LIN {X 0,Y 354.82,Z 396.284,A -85,B 0,C 180,E1 -13539.425,E2 -13539.425} C_VEL
LIN {X 0,Y 354.8,Z 396.287,A -85,B 0,C 180,E1 -13542.871,E2 -13542.871} C_VEL
LIN {X 0,Y 354.764,Z 396.297,A -85,B 0,C 180,E1 -13546.105,E2 -13546.105} C_VEL
LIN {X 0,Y 354.786,Z 396.288,A -85,B 0,C 180,E1 -13549.18,E2 -13549.18} C_VEL
LIN {X 0,Y 354.807,Z 396.289,A -85,B 0,C 180,E1 -13552.403,E2 -13552.403} C_VEL
LIN {X 0,Y 354.811,Z 396.285,A -85,B 0,C 180,E1 -13554.942,E2 -13554.942} C_VEL
LIN {X 0,Y 354.793,Z 396.29,A -85,B 0,C 180,E1 -13558.406,E2 -13558.406} C_VEL
LIN {X 0,Y 354.847,Z 396.283,A -85,B 0,C 180,E1 -13561.62,E2 -13561.62} C_VEL
LIN {X 0,Y 354.9,Z 396.278,A -85,B 0,C 180,E1 -13564.174,E2 -13564.174} C_VEL
LIN {X 0,Y 354.836,Z 396.288,A -85,B 0,C 180,E1 -13567.895,E2 -13567.895} C_VEL
LIN {X 0,Y 354.925,Z 396.277,A -85,B 0,C 180,E1 -13571.892,E2 -13571.892} C_VEL
LIN {X 0,Y 354.945,Z 396.274,A -85,B 0,C 180,E1 -13575.982,E2 -13575.982} C_VEL
LIN {X 0,Y 354.981,Z 396.27,A -85,B 0,C 180,E1 -13579.736,E2 -13579.736} C_VEL
LIN {X 0,Y 355.117,Z 396.251,A -85,B 0,C 180,E1 -13582.037,E2 -13582.037} C_VEL
LIN {X 0,Y 355.095,Z 396.251,A -85,B 0,C 180,E1 -13584.321,E2 -13584.321} C_VEL
LIN {X 0,Y 355.123,Z 396.247,A -85,B 0,C 180,E1 -13588.866,E2 -13588.866} C_VEL
LIN {X 0,Y 354.261,Z 396.361,A -85,B 0,C 180,E1 -13591.137,E2 -13591.137} C_VEL
LIN {X 0,Y 354.367,Z 399.159,A -85,B 0,C 180,E1 -13594.55,E2 -13594.55} C_VEL
LIN {X 0,Y 354.171,Z 402.38,A -85,B 0,C 180,E1 -13597.985,E2 -13597.985} C_VEL
LIN {X 0,Y 353.989,Z 406.197,A -85,B 0,C 180,E1 -13601.887,E2 -13601.887} C_VEL
LIN {X 0,Y 357.569,Z 419.481,A -85,B 0,C 180,E1 -13602.63,E2 -13602.63} C_VEL
LIN {X 0,Y 360.42,Z 432.028,A -85,B 0,C 180,E1 -13603.532,E2 -13603.532} C_VEL
LIN {X 0,Y 360.675,Z 435.61,A -85,B 0,C 180,E1 -13603.81,E2 -13603.81} C_VEL
LIN {X 0,Y 359.83,Z 446.641,A -85,B 0,C 180,E1 -13604.709,E2 -13604.709} C_VEL
LIN {X 0,Y 358.918,Z 456.939,A -85,B 0,C 180,E1 -13605.765,E2 -13605.765} C_VEL
LIN {X 0,Y 357.825,Z 467.606,A -85,B 0,C 180,E1 -13607.134,E2 -13607.134} C_VEL
LIN {X 0,Y 356.806,Z 477.084,A -85,B 0,C 180,E1 -13608.646,E2 -13608.646} C_VEL
LIN {X 0,Y 355.86,Z 485.097,A -85,B 0,C 180,E1 -13610.219,E2 -13610.219} C_VEL
LIN {X 0,Y 355.001,Z 492.665,A -85,B 0,C 180,E1 -13612.095,E2 -13612.095} C_VEL
LIN {X 0,Y 354.467,Z 497.998,A -85,B 0,C 180,E1 -13613.763,E2 -13613.763} C_VEL
LIN {X 0,Y 353.942,Z 503.231,A -85,B 0,C 180,E1 -13615.902,E2 -13615.902} C_VEL
LIN {X 0,Y 353.764,Z 505.535,A -85,B 0,C 180,E1 -13617.189,E2 -13617.189} C_VEL
LIN {X 0,Y 353.425,Z 507.859,A -85,B 0,C 180,E1 -13618.959,E2 -13618.959} C_VEL
LIN {X 0,Y 353.286,Z 509.399,A -85,B 0,C 180,E1 -13621.194,E2 -13621.194} C_VEL
LIN {X 0,Y 353.305,Z 509.409,A -85,B 0,C 180,E1 -13623.334,E2 -13623.334} C_VEL
LIN {X 0,Y 353.494,Z 508.102,A -85,B 0,C 180,E1 -13625.398,E2 -13625.398} C_VEL
LIN {X 0,Y 353.871,Z 505.571,A -85,B 0,C 180,E1 -13627.399,E2 -13627.399} C_VEL
LIN {X 0,Y 354.373,Z 501.731,A -85,B 0,C 180,E1 -13629.392,E2 -13629.392} C_VEL
LIN {X 0,Y 354.911,Z 496.973,A -85,B 0,C 180,E1 -13631.194,E2 -13631.194} C_VEL
LIN {X 0,Y 355.686,Z 490.73,A -85,B 0,C 180,E1 -13633.022,E2 -13633.022} C_VEL
LIN {X 0,Y 356.677,Z 482.905,A -85,B 0,C 180,E1 -13634.832,E2 -13634.832} C_VEL
LIN {X 0,Y 356.532,Z 479.281,A -85,B 0,C 180,E1 -13635.576,E2 -13635.576} C_VEL
LIN {X 0,Y 354.521,Z 473.127,A -85,B 0,C 180,E1 -13636.799,E2 -13636.799} C_VEL
LIN {X 0,Y 352.549,Z 466.534,A -85,B 0,C 180,E1 -13637.955,E2 -13637.955} C_VEL
LIN {X 0,Y 352.45,Z 462.072,A -85,B 0,C 180,E1 -13638.582,E2 -13638.582} C_VEL
LIN {X 0,Y 353.487,Z 452.087,A -85,B 0,C 180,E1 -13639.726,E2 -13639.726} C_VEL
LIN {X 0,Y 354.57,Z 440.766,A -85,B 0,C 180,E1 -13640.757,E2 -13640.757} C_VEL
LIN {X 0,Y 354.763,Z 436.437,A -85,B 0,C 180,E1 -13641.097,E2 -13641.097} C_VEL
LIN {X 0,Y 352.322,Z 425.509,A -85,B 0,C 180,E1 -13642.011,E2 -13642.011} C_VEL
LIN {X 0,Y 348.485,Z 412.951,A -85,B 0,C 180,E1 -13642.905,E2 -13642.905} C_VEL
LIN {X 0,Y 346.967,Z 408.125,A -85,B 0,C 180,E1 -13643.215,E2 -13643.215} C_VEL
LIN {X 0,Y 347.163,Z 405.007,A -85,B 0,C 180,E1 -13646.866,E2 -13646.866} C_VEL
LIN {X 0,Y 347.352,Z 402.017,A -85,B 0,C 180,E1 -13650.46,E2 -13650.46} C_VEL
LIN {X 0,Y 347.472,Z 399.497,A -85,B 0,C 180,E1 -13653.578,E2 -13653.578} C_VEL
LIN {X 0,Y 347.611,Z 397.471,A -85,B 0,C 180,E1 -13656.149,E2 -13656.149} C_VEL
LIN {X 0,Y 347.759,Z 397.173,A -85,B 0,C 180,E1 -13658.668,E2 -13658.668} C_VEL
LIN {X 0,Y 347.862,Z 397.155,A -85,B 0,C 180,E1 -13662.359,E2 -13662.359} C_VEL
LIN {X 0,Y 347.894,Z 397.153,A -85,B 0,C 180,E1 -13665.97,E2 -13665.97} C_VEL
LIN {X 0,Y 347.924,Z 397.149,A -85,B 0,C 180,E1 -13669.525,E2 -13669.525} C_VEL
LIN {X 0,Y 348.087,Z 397.126,A -85,B 0,C 180,E1 -13673.042,E2 -13673.042} C_VEL
LIN {X 0,Y 348.203,Z 397.11,A -85,B 0,C 180,E1 -13677.686,E2 -13677.686} C_VEL
LIN {X 0,Y 348.341,Z 397.092,A -85,B 0,C 180,E1 -13680,E2 -13680} C_VEL
LIN {X 0,Y 348.203,Z 397.109,A -85,B 0,C 180,E1 -13682.313,E2 -13682.313} C_VEL
LIN {X 0,Y 348.087,Z 397.127,A -85,B 0,C 180,E1 -13686.958,E2 -13686.958} C_VEL
LIN {X 0,Y 347.924,Z 397.143,A -85,B 0,C 180,E1 -13690.474,E2 -13690.474} C_VEL
LIN {X 0,Y 347.894,Z 397.15,A -85,B 0,C 180,E1 -13694.15,E2 -13694.15} C_VEL
LIN {X 0,Y 347.887,Z 397.15,A -85,B 0,C 180,E1 -13698.291,E2 -13698.291} C_VEL
LIN {X 0,Y 347.784,Z 397.165,A -85,B 0,C 180,E1 -13701.635,E2 -13701.635} C_VEL
LIN {X 0,Y 347.808,Z 397.162,A -85,B 0,C 180,E1 -13705.109,E2 -13705.109} C_VEL
LIN {X 0,Y 347.804,Z 397.163,A -85,B 0,C 180,E1 -13707.694,E2 -13707.694} C_VEL
LIN {X 0,Y 347.745,Z 397.172,A -85,B 0,C 180,E1 -13710.348,E2 -13710.348} C_VEL
LIN {X 0,Y 347.745,Z 397.174,A -85,B 0,C 180,E1 -13714.044,E2 -13714.044} C_VEL
LIN {X 0,Y 347.76,Z 397.17,A -85,B 0,C 180,E1 -13717.321,E2 -13717.321} C_VEL
LIN {X 0,Y 347.753,Z 397.169,A -85,B 0,C 180,E1 -13720.294,E2 -13720.294} C_VEL
LIN {X 0,Y 347.79,Z 397.314,A -85,B 0,C 180,E1 -13721.824,E2 -13721.824} C_VEL
LIN {X 0,Y 348.52,Z 401.454,A -85,B 0,C 180,E1 -13725.108,E2 -13725.108} C_VEL
LIN {X 0,Y 349.367,Z 406.016,A -85,B 0,C 180,E1 -13728.407,E2 -13728.407} C_VEL
LIN {X 0,Y 350.163,Z 410.733,A -85,B 0,C 180,E1 -13731.524,E2 -13731.524} C_VEL
LIN {X 0,Y 350.496,Z 413.638,A -85,B 0,C 180,E1 -13733.328,E2 -13733.328} C_VEL
LIN {X 0,Y 350.032,Z 417.928,A -85,B 0,C 180,E1 -13735.793,E2 -13735.793} C_VEL
LIN {X 0,Y 349.088,Z 425.333,A -85,B 0,C 180,E1 -13739.781,E2 -13739.781} C_VEL
LIN {X 0,Y 348.231,Z 432.827,A -85,B 0,C 180,E1 -13743.641,E2 -13743.641} C_VEL
LIN {X 0,Y 347.569,Z 440.436,A -85,B 0,C 180,E1 -13747.407,E2 -13747.407} C_VEL
LIN {X 0,Y 347.384,Z 443.37,A -85,B 0,C 180,E1 -13748.844,E2 -13748.844} C_VEL
LIN {X 0,Y 350.074,Z 457.101,A -85,B 0,C 180,E1 -13749.538,E2 -13749.538} C_VEL
LIN {X 0,Y 351.773,Z 470.332,A -85,B 0,C 180,E1 -13750.4,E2 -13750.4} C_VEL
LIN {X 0,Y 352.9,Z 482.718,A -85,B 0,C 180,E1 -13751.419,E2 -13751.419} C_VEL
LIN {X 0,Y 352.517,Z 489.14,A -85,B 0,C 180,E1 -13752,E2 -13752} C_VEL
LIN {X 0,Y 351.116,Z 500.982,A -85,B 0,C 180,E1 -13753.278,E2 -13753.278} C_VEL
LIN {X 0,Y 350.038,Z 510.242,A -85,B 0,C 180,E1 -13754.523,E2 -13754.523} C_VEL
LIN {X 0,Y 349.027,Z 519.346,A -85,B 0,C 180,E1 -13756.017,E2 -13756.017} C_VEL
LIN {X 0,Y 347.998,Z 527.91,A -85,B 0,C 180,E1 -13757.757,E2 -13757.757} C_VEL
LIN {X 0,Y 347.282,Z 534.815,A -85,B 0,C 180,E1 -13759.506,E2 -13759.506} C_VEL
LIN {X 0,Y 346.735,Z 540.361,A -85,B 0,C 180,E1 -13761.256,E2 -13761.256} C_VEL
LIN {X 0,Y 346.419,Z 544.723,A -85,B 0,C 180,E1 -13763.008,E2 -13763.008} C_VEL
LIN {X 0,Y 346.318,Z 547.047,A -85,B 0,C 180,E1 -13764.176,E2 -13764.176} C_VEL
LIN {X 0,Y 346.271,Z 548.911,A -85,B 0,C 180,E1 -13765.343,E2 -13765.343} C_VEL
LIN {X 0,Y 346.223,Z 551.331,A -85,B 0,C 180,E1 -13767.673,E2 -13767.673} C_VEL
LIN {X 0,Y 346.32,Z 551.953,A -85,B 0,C 180,E1 -13768.837,E2 -13768.837} C_VEL
LIN {X 0,Y 346.35,Z 552.148,A -85,B 0,C 180,E1 -13770,E2 -13770} C_VEL
LIN {X 0,Y 346.339,Z 551.916,A -85,B 0,C 180,E1 -13771.162,E2 -13771.162} C_VEL
LIN {X 0,Y 346.206,Z 550.263,A -85,B 0,C 180,E1 -13773.491,E2 -13773.491} C_VEL
LIN {X 0,Y 346.274,Z 548.811,A -85,B 0,C 180,E1 -13774.656,E2 -13774.656} C_VEL
LIN {X 0,Y 346.344,Z 546.358,A -85,B 0,C 180,E1 -13776.116,E2 -13776.116} C_VEL
LIN {X 0,Y 346.591,Z 541.732,A -85,B 0,C 180,E1 -13778.16,E2 -13778.16} C_VEL
LIN {X 0,Y 347.171,Z 535.476,A -85,B 0,C 180,E1 -13780.202,E2 -13780.202} C_VEL
LIN {X 0,Y 347.811,Z 528.66,A -85,B 0,C 180,E1 -13781.953,E2 -13781.953} C_VEL
LIN {X 0,Y 348.832,Z 520.203,A -85,B 0,C 180,E1 -13783.693,E2 -13783.693} C_VEL
LIN {X 0,Y 349.955,Z 510.721,A -85,B 0,C 180,E1 -13785.251,E2 -13785.251} C_VEL
LIN {X 0,Y 350.873,Z 500.782,A -85,B 0,C 180,E1 -13786.584,E2 -13786.584} C_VEL
LIN {X 0,Y 352.108,Z 490.179,A -85,B 0,C 180,E1 -13787.721,E2 -13787.721} C_VEL
LIN {X 0,Y 352.687,Z 483.789,A -85,B 0,C 180,E1 -13788.291,E2 -13788.291} C_VEL
LIN {X 0,Y 351.491,Z 471.586,A -85,B 0,C 180,E1 -13789.281,E2 -13789.281} C_VEL
LIN {X 0,Y 349.823,Z 458.882,A -85,B 0,C 180,E1 -13790.094,E2 -13790.094} C_VEL
LIN {X 0,Y 347.566,Z 446.078,A -85,B 0,C 180,E1 -13790.71,E2 -13790.71} C_VEL
LIN {X 0,Y 347.366,Z 444.386,A -85,B 0,C 180,E1 -13790.813,E2 -13790.813} C_VEL
LIN {X 0,Y 347.975,Z 436.534,A -85,B 0,C 180,E1 -13794.652,E2 -13794.652} C_VEL
LIN {X 0,Y 348.662,Z 429.282,A -85,B 0,C 180,E1 -13798.273,E2 -13798.273} C_VEL
LIN {X 0,Y 349.314,Z 422.946,A -85,B 0,C 180,E1 -13801.54,E2 -13801.54} C_VEL
LIN {X 0,Y 350.133,Z 417.113,A -85,B 0,C 180,E1 -13804.617,E2 -13804.617} C_VEL
LIN {X 0,Y 350.477,Z 412.823,A -85,B 0,C 180,E1 -13806.982,E2 -13806.982} C_VEL
LIN {X 0,Y 349.931,Z 408.97,A -85,B 0,C 180,E1 -13809.243,E2 -13809.243} C_VEL
LIN {X 0,Y 348.909,Z 403.557,A -85,B 0,C 180,E1 -13812.619,E2 -13812.619} C_VEL
LIN {X 0,Y 348.055,Z 398.681,A -85,B 0,C 180,E1 -13815.843,E2 -13815.843} C_VEL
LIN {X 0,Y 347.778,Z 397.166,A -85,B 0,C 180,E1 -13817.036,E2 -13817.036} C_VEL
LIN {X 0,Y 347.761,Z 397.168,A -85,B 0,C 180,E1 -13821.208,E2 -13821.208} C_VEL
LIN {X 0,Y 347.783,Z 397.161,A -85,B 0,C 180,E1 -13824.124,E2 -13824.124} C_VEL
LIN {X 0,Y 347.732,Z 397.167,A -85,B 0,C 180,E1 -13828.086,E2 -13828.086} C_VEL
LIN {X 0,Y 347.772,Z 397.167,A -85,B 0,C 180,E1 -13830.987,E2 -13830.987} C_VEL
LIN {X 0,Y 347.824,Z 397.156,A -85,B 0,C 180,E1 -13833.607,E2 -13833.607} C_VEL
LIN {X 0,Y 347.781,Z 397.161,A -85,B 0,C 180,E1 -13836.161,E2 -13836.161} C_VEL
LIN {X 0,Y 347.805,Z 397.158,A -85,B 0,C 180,E1 -13839.909,E2 -13839.909} C_VEL
LIN {X 0,Y 347.858,Z 397.153,A -85,B 0,C 180,E1 -13842.359,E2 -13842.359} C_VEL
LIN {X 0,Y 347.89,Z 397.147,A -85,B 0,C 180,E1 -13845.971,E2 -13845.971} C_VEL
LIN {X 0,Y 347.921,Z 397.144,A -85,B 0,C 180,E1 -13849.525,E2 -13849.525} C_VEL
LIN {X 0,Y 348.084,Z 397.126,A -85,B 0,C 180,E1 -13853.042,E2 -13853.042} C_VEL
LIN {X 0,Y 348.2,Z 397.109,A -85,B 0,C 180,E1 -13857.687,E2 -13857.687} C_VEL
LIN {X 0,Y 348.36,Z 397.09,A -85,B 0,C 180,E1 -13860,E2 -13860} C_VEL
LIN {X 0,Y 348.2,Z 397.112,A -85,B 0,C 180,E1 -13862.314,E2 -13862.314} C_VEL
LIN {X 0,Y 348.098,Z 397.124,A -85,B 0,C 180,E1 -13866.958,E2 -13866.958} C_VEL
LIN {X 0,Y 347.96,Z 397.139,A -85,B 0,C 180,E1 -13869.299,E2 -13869.299} C_VEL
LIN {X 0,Y 347.882,Z 397.151,A -85,B 0,C 180,E1 -13872.84,E2 -13872.84} C_VEL
LIN {X 0,Y 347.832,Z 397.16,A -85,B 0,C 180,E1 -13876.432,E2 -13876.432} C_VEL
LIN {X 0,Y 347.849,Z 397.154,A -85,B 0,C 180,E1 -13878.861,E2 -13878.861} C_VEL
LIN {X 0,Y 347.767,Z 397.167,A -85,B 0,C 180,E1 -13882.58,E2 -13882.58} C_VEL
LIN {X 0,Y 347.806,Z 397.158,A -85,B 0,C 180,E1 -13885.109,E2 -13885.109} C_VEL
LIN {X 0,Y 347.805,Z 397.159,A -85,B 0,C 180,E1 -13887.695,E2 -13887.695} C_VEL
LIN {X 0,Y 347.758,Z 397.169,A -85,B 0,C 180,E1 -13890.347,E2 -13890.347} C_VEL
LIN {X 0,Y 347.739,Z 397.17,A -85,B 0,C 180,E1 -13894.465,E2 -13894.465} C_VEL
LIN {X 0,Y 347.772,Z 397.166,A -85,B 0,C 180,E1 -13897.99,E2 -13897.99} C_VEL
LIN {X 0,Y 347.763,Z 397.166,A -85,B 0,C 180,E1 -13901.829,E2 -13901.829} C_VEL
LIN {X 0,Y 347.704,Z 397.17,A -85,B 0,C 180,E1 -13905.027,E2 -13905.027} C_VEL
LIN {X 0,Y 347.748,Z 397.168,A -85,B 0,C 180,E1 -13908.398,E2 -13908.398} C_VEL
LIN {X 0,Y 347.773,Z 397.167,A -85,B 0,C 180,E1 -13912.012,E2 -13912.012} C_VEL
LIN {X 0,Y 347.743,Z 397.167,A -85,B 0,C 180,E1 -13915.537,E2 -13915.537} C_VEL
LIN {X 0,Y 347.745,Z 397.169,A -85,B 0,C 180,E1 -13918.301,E2 -13918.301} C_VEL
LIN {X 0,Y 347.778,Z 397.161,A -85,B 0,C 180,E1 -13920.989,E2 -13920.989} C_VEL
LIN {X 0,Y 347.832,Z 397.157,A -85,B 0,C 180,E1 -13923.609,E2 -13923.609} C_VEL
LIN {X 0,Y 347.79,Z 397.164,A -85,B 0,C 180,E1 -13926.163,E2 -13926.163} C_VEL
LIN {X 0,Y 347.819,Z 397.162,A -85,B 0,C 180,E1 -13929.91,E2 -13929.91} C_VEL
LIN {X 0,Y 347.869,Z 397.152,A -85,B 0,C 180,E1 -13932.36,E2 -13932.36} C_VEL
LIN {X 0,Y 347.9,Z 397.151,A -85,B 0,C 180,E1 -13935.971,E2 -13935.971} C_VEL
LIN {X 0,Y 347.931,Z 397.145,A -85,B 0,C 180,E1 -13939.526,E2 -13939.526} C_VEL
LIN {X 0,Y 348.078,Z 397.129,A -85,B 0,C 180,E1 -13941.875,E2 -13941.875} C_VEL
LIN {X 0,Y 348.07,Z 397.127,A -85,B 0,C 180,E1 -13944.206,E2 -13944.206} C_VEL
LIN {X 0,Y 348.091,Z 397.122,A -85,B 0,C 180,E1 -13948.843,E2 -13948.843} C_VEL
LIN {X 0,Y 347.206,Z 397.239,A -85,B 0,C 180,E1 -13951.16,E2 -13951.16} C_VEL
LIN {X 0,Y 347.316,Z 400.101,A -85,B 0,C 180,E1 -13954.643,E2 -13954.643} C_VEL
LIN {X 0,Y 347.111,Z 403.298,A -85,B 0,C 180,E1 -13958.148,E2 -13958.148} C_VEL
LIN {X 0,Y 346.894,Z 406.47,A -85,B 0,C 180,E1 -13961.467,E2 -13961.467} C_VEL
LIN {X 0,Y 350.716,Z 420.405,A -85,B 0,C 180,E1 -13962.293,E2 -13962.293} C_VEL
LIN {X 0,Y 353.52,Z 432.875,A -85,B 0,C 180,E1 -13963.216,E2 -13963.216} C_VEL
LIN {X 0,Y 353.9,Z 436.266,A -85,B 0,C 180,E1 -13963.494,E2 -13963.494} C_VEL
LIN {X 0,Y 353.014,Z 447.259,A -85,B 0,C 180,E1 -13964.41,E2 -13964.41} C_VEL
LIN {X 0,Y 351.922,Z 458.801,A -85,B 0,C 180,E1 -13965.64,E2 -13965.64} C_VEL
LIN {X 0,Y 350.819,Z 468.918,A -85,B 0,C 180,E1 -13966.992,E2 -13966.992} C_VEL
LIN {X 0,Y 349.859,Z 477.746,A -85,B 0,C 180,E1 -13968.444,E2 -13968.444} C_VEL
LIN {X 0,Y 348.897,Z 485.606,A -85,B 0,C 180,E1 -13970.025,E2 -13970.025} C_VEL
LIN {X 0,Y 348.058,Z 492.489,A -85,B 0,C 180,E1 -13971.745,E2 -13971.745} C_VEL
LIN {X 0,Y 347.531,Z 497.324,A -85,B 0,C 180,E1 -13973.225,E2 -13973.225} C_VEL
LIN {X 0,Y 346.998,Z 502.312,A -85,B 0,C 180,E1 -13975.171,E2 -13975.171} C_VEL
LIN {X 0,Y 346.738,Z 505.624,A -85,B 0,C 180,E1 -13976.895,E2 -13976.895} C_VEL
LIN {X 0,Y 346.321,Z 508.605,A -85,B 0,C 180,E1 -13979.236,E2 -13979.236} C_VEL
LIN {X 0,Y 346.208,Z 509.906,A -85,B 0,C 180,E1 -13981.504,E2 -13981.504} C_VEL
LIN {X 0,Y 346.232,Z 509.74,A -85,B 0,C 180,E1 -13983.67,E2 -13983.67} C_VEL
LIN {X 0,Y 346.525,Z 508.021,A -85,B 0,C 180,E1 -13986.026,E2 -13986.026} C_VEL
LIN {X 0,Y 346.898,Z 505.598,A -85,B 0,C 180,E1 -13987.802,E2 -13987.802} C_VEL
LIN {X 0,Y 347.388,Z 501.733,A -85,B 0,C 180,E1 -13989.755,E2 -13989.755} C_VEL
LIN {X 0,Y 348.058,Z 496.267,A -85,B 0,C 180,E1 -13991.784,E2 -13991.784} C_VEL
LIN {X 0,Y 349.014,Z 489.379,A -85,B 0,C 180,E1 -13993.74,E2 -13993.74} C_VEL
LIN {X 0,Y 349.993,Z 482.21,A -85,B 0,C 180,E1 -13995.346,E2 -13995.346} C_VEL
LIN {X 0,Y 351.09,Z 473.823,A -85,B 0,C 180,E1 -13996.876,E2 -13996.876} C_VEL
LIN {X 0,Y 352.297,Z 463.334,A -85,B 0,C 180,E1 -13998.424,E2 -13998.424} C_VEL
LIN {X 0,Y 352.45,Z 462.072,A -85,B 0,C 180,E1 -13998.582,E2 -13998.582} C_VEL
LIN {X 0,Y 352.394,Z 455.899,A -85,B 0,C 180,E1 -13999.362,E2 -13999.362} C_VEL
LIN {X 0,Y 351.186,Z 449.734,A -85,B 0,C 180,E1 -14000.13,E2 -14000.13} C_VEL
LIN {X 0,Y 349.464,Z 443.357,A -85,B 0,C 180,E1 -14000.867,E2 -14000.867} C_VEL
LIN {X 0,Y 347.859,Z 436.701,A -85,B 0,C 180,E1 -14001.543,E2 -14001.543} C_VEL
LIN {X 0,Y 345.286,Z 425.748,A -85,B 0,C 180,E1 -14002.489,E2 -14002.489} C_VEL
LIN {X 0,Y 341.446,Z 413.364,A -85,B 0,C 180,E1 -14003.4,E2 -14003.4} C_VEL
LIN {X 0,Y 339.942,Z 408.589,A -85,B 0,C 180,E1 -14003.734,E2 -14003.734} C_VEL
LIN {X 0,Y 340.147,Z 405.423,A -85,B 0,C 180,E1 -14007.506,E2 -14007.506} C_VEL
LIN {X 0,Y 340.306,Z 403.155,A -85,B 0,C 180,E1 -14010.287,E2 -14010.287} C_VEL
LIN {X 0,Y 340.436,Z 401.017,A -85,B 0,C 180,E1 -14012.988,E2 -14012.988} C_VEL
LIN {X 0,Y 340.612,Z 398.955,A -85,B 0,C 180,E1 -14015.627,E2 -14015.627} C_VEL
LIN {X 0,Y 340.58,Z 398.068,A -85,B 0,C 180,E1 -14016.916,E2 -14016.916} C_VEL
LIN {X 0,Y 340.782,Z 398.039,A -85,B 0,C 180,E1 -14020.733,E2 -14020.733} C_VEL
LIN {X 0,Y 340.782,Z 398.038,A -85,B 0,C 180,E1 -14023.218,E2 -14023.218} C_VEL
LIN {X 0,Y 340.84,Z 398.03,A -85,B 0,C 180,E1 -14026.89,E2 -14026.89} C_VEL
LIN {X 0,Y 340.91,Z 398.02,A -85,B 0,C 180,E1 -14030.507,E2 -14030.507} C_VEL
LIN {X 0,Y 341.055,Z 398.001,A -85,B 0,C 180,E1 -14032.898,E2 -14032.898} C_VEL
LIN {X 0,Y 341.165,Z 397.986,A -85,B 0,C 180,E1 -14037.639,E2 -14037.639} C_VEL
LIN {X 0,Y 341.291,Z 397.97,A -85,B 0,C 180,E1 -14040,E2 -14040} C_VEL
LIN {X 0,Y 341.165,Z 397.986,A -85,B 0,C 180,E1 -14042.361,E2 -14042.361} C_VEL
LIN {X 0,Y 341.055,Z 398.003,A -85,B 0,C 180,E1 -14047.102,E2 -14047.102} C_VEL
LIN {X 0,Y 340.866,Z 398.022,A -85,B 0,C 180,E1 -14050.694,E2 -14050.694} C_VEL
LIN {X 0,Y 340.859,Z 398.026,A -85,B 0,C 180,E1 -14054.325,E2 -14054.325} C_VEL
LIN {X 0,Y 340.834,Z 398.027,A -85,B 0,C 180,E1 -14058.467,E2 -14058.467} C_VEL
LIN {X 0,Y 340.75,Z 398.042,A -85,B 0,C 180,E1 -14061.857,E2 -14061.857} C_VEL
LIN {X 0,Y 340.768,Z 398.039,A -85,B 0,C 180,E1 -14065.665,E2 -14065.665} C_VEL
LIN {X 0,Y 340.725,Z 398.043,A -85,B 0,C 180,E1 -14068.321,E2 -14068.321} C_VEL
LIN {X 0,Y 340.694,Z 398.047,A -85,B 0,C 180,E1 -14071.045,E2 -14071.045} C_VEL
LIN {X 0,Y 340.715,Z 398.047,A -85,B 0,C 180,E1 -14075.279,E2 -14075.279} C_VEL
LIN {X 0,Y 340.715,Z 398.047,A -85,B 0,C 180,E1 -14078.388,E2 -14078.388} C_VEL
LIN {X 0,Y 340.724,Z 398.137,A -85,B 0,C 180,E1 -14081.159,E2 -14081.159} C_VEL
LIN {X 0,Y 341.408,Z 402.065,A -85,B 0,C 180,E1 -14084.419,E2 -14084.419} C_VEL
LIN {X 0,Y 342.238,Z 406.375,A -85,B 0,C 180,E1 -14087.67,E2 -14087.67} C_VEL
LIN {X 0,Y 343.082,Z 411.395,A -85,B 0,C 180,E1 -14091.117,E2 -14091.117} C_VEL
LIN {X 0,Y 343.476,Z 414.258,A -85,B 0,C 180,E1 -14092.939,E2 -14092.939} C_VEL
LIN {X 0,Y 343.222,Z 417.737,A -85,B 0,C 180,E1 -14095.017,E2 -14095.017} C_VEL
LIN {X 0,Y 342.181,Z 425.051,A -85,B 0,C 180,E1 -14099.105,E2 -14099.105} C_VEL
LIN {X 0,Y 341.275,Z 432.497,A -85,B 0,C 180,E1 -14103.06,E2 -14103.06} C_VEL
LIN {X 0,Y 340.547,Z 440.057,A -85,B 0,C 180,E1 -14106.914,E2 -14106.914} C_VEL
LIN {X 0,Y 340.373,Z 443.137,A -85,B 0,C 180,E1 -14108.351,E2 -14108.351} C_VEL
LIN {X 0,Y 343.09,Z 456.301,A -85,B 0,C 180,E1 -14109.044,E2 -14109.044} C_VEL
LIN {X 0,Y 344.841,Z 469.313,A -85,B 0,C 180,E1 -14109.915,E2 -14109.915} C_VEL
LIN {X 0,Y 345.836,Z 481.465,A -85,B 0,C 180,E1 -14110.927,E2 -14110.927} C_VEL
LIN {X 0,Y 346.083,Z 485.84,A -85,B 0,C 180,E1 -14111.347,E2 -14111.347} C_VEL
LIN {X 0,Y 344.767,Z 497.117,A -85,B 0,C 180,E1 -14112.502,E2 -14112.502} C_VEL
LIN {X 0,Y 343.435,Z 507.636,A -85,B 0,C 180,E1 -14113.856,E2 -14113.856} C_VEL
LIN {X 0,Y 342.32,Z 517.398,A -85,B 0,C 180,E1 -14115.434,E2 -14115.434} C_VEL
LIN {X 0,Y 341.198,Z 526.29,A -85,B 0,C 180,E1 -14117.207,E2 -14117.207} C_VEL
LIN {X 0,Y 340.342,Z 533.432,A -85,B 0,C 180,E1 -14118.988,E2 -14118.988} C_VEL
LIN {X 0,Y 339.697,Z 539.99,A -85,B 0,C 180,E1 -14121.073,E2 -14121.073} C_VEL
LIN {X 0,Y 339.347,Z 544.336,A -85,B 0,C 180,E1 -14122.862,E2 -14122.862} C_VEL
LIN {X 0,Y 339.238,Z 546.652,A -85,B 0,C 180,E1 -14124.054,E2 -14124.054} C_VEL
LIN {X 0,Y 339.189,Z 548.503,A -85,B 0,C 180,E1 -14125.246,E2 -14125.246} C_VEL
LIN {X 0,Y 339.13,Z 549.906,A -85,B 0,C 180,E1 -14126.435,E2 -14126.435} C_VEL
LIN {X 0,Y 339.227,Z 551.529,A -85,B 0,C 180,E1 -14128.813,E2 -14128.813} C_VEL
LIN {X 0,Y 339.29,Z 551.716,A -85,B 0,C 180,E1 -14130,E2 -14130} C_VEL
LIN {X 0,Y 339.26,Z 551.478,A -85,B 0,C 180,E1 -14131.187,E2 -14131.187} C_VEL
LIN {X 0,Y 339.13,Z 549.815,A -85,B 0,C 180,E1 -14133.564,E2 -14133.564} C_VEL
LIN {X 0,Y 339.193,Z 548.35,A -85,B 0,C 180,E1 -14134.754,E2 -14134.754} C_VEL
LIN {X 0,Y 339.298,Z 545.331,A -85,B 0,C 180,E1 -14136.541,E2 -14136.541} C_VEL
LIN {X 0,Y 339.547,Z 541.243,A -85,B 0,C 180,E1 -14138.33,E2 -14138.33} C_VEL
LIN {X 0,Y 340.14,Z 534.965,A -85,B 0,C 180,E1 -14140.415,E2 -14140.415} C_VEL
LIN {X 0,Y 340.841,Z 528.126,A -85,B 0,C 180,E1 -14142.201,E2 -14142.201} C_VEL
LIN {X 0,Y 341.877,Z 519.627,A -85,B 0,C 180,E1 -14143.977,E2 -14143.977} C_VEL
LIN {X 0,Y 342.966,Z 510.886,A -85,B 0,C 180,E1 -14145.449,E2 -14145.449} C_VEL
LIN {X 0,Y 344.051,Z 500.125,A -85,B 0,C 180,E1 -14146.922,E2 -14146.922} C_VEL
LIN {X 0,Y 345.309,Z 489.46,A -85,B 0,C 180,E1 -14148.081,E2 -14148.081} C_VEL
LIN {X 0,Y 345.774,Z 484.738,A -85,B 0,C 180,E1 -14148.516,E2 -14148.516} C_VEL
LIN {X 0,Y 344.735,Z 473.294,A -85,B 0,C 180,E1 -14149.498,E2 -14149.498} C_VEL
LIN {X 0,Y 342.999,Z 459.609,A -85,B 0,C 180,E1 -14150.42,E2 -14150.42} C_VEL
LIN {X 0,Y 340.7,Z 446.287,A -85,B 0,C 180,E1 -14151.098,E2 -14151.098} C_VEL
LIN {X 0,Y 340.338,Z 444.086,A -85,B 0,C 180,E1 -14151.184,E2 -14151.184} C_VEL
LIN {X 0,Y 340.936,Z 436.673,A -85,B 0,C 180,E1 -14154.905,E2 -14154.905} C_VEL
LIN {X 0,Y 341.732,Z 428.894,A -85,B 0,C 180,E1 -14158.9,E2 -14158.9} C_VEL
LIN {X 0,Y 342.608,Z 421.612,A -85,B 0,C 180,E1 -14162.749,E2 -14162.749} C_VEL
LIN {X 0,Y 343.357,Z 416.262,A -85,B 0,C 180,E1 -14165.685,E2 -14165.685} C_VEL
LIN {X 0,Y 343.317,Z 412.438,A -85,B 0,C 180,E1 -14167.887,E2 -14167.887} C_VEL
LIN {X 0,Y 342.41,Z 407.302,A -85,B 0,C 180,E1 -14171.055,E2 -14171.055} C_VEL
LIN {X 0,Y 341.474,Z 402.196,A -85,B 0,C 180,E1 -14174.407,E2 -14174.407} C_VEL
LIN {X 0,Y 340.731,Z 398.044,A -85,B 0,C 180,E1 -14177.342,E2 -14177.342} C_VEL
LIN {X 0,Y 340.705,Z 398.046,A -85,B 0,C 180,E1 -14180.248,E2 -14180.248} C_VEL
LIN {X 0,Y 340.705,Z 398.043,A -85,B 0,C 180,E1 -14183.558,E2 -14183.558} C_VEL
LIN {X 0,Y 340.686,Z 398.045,A -85,B 0,C 180,E1 -14186.153,E2 -14186.153} C_VEL
LIN {X 0,Y 340.735,Z 398.039,A -85,B 0,C 180,E1 -14190.329,E2 -14190.329} C_VEL
LIN {X 0,Y 340.796,Z 398.035,A -85,B 0,C 180,E1 -14193.019,E2 -14193.019} C_VEL
LIN {X 0,Y 340.749,Z 398.037,A -85,B 0,C 180,E1 -14195.638,E2 -14195.638} C_VEL
LIN {X 0,Y 340.745,Z 398.038,A -85,B 0,C 180,E1 -14199.474,E2 -14199.474} C_VEL
LIN {X 0,Y 340.85,Z 398.024,A -85,B 0,C 180,E1 -14201.984,E2 -14201.984} C_VEL
LIN {X 0,Y 340.862,Z 398.022,A -85,B 0,C 180,E1 -14205.705,E2 -14205.705} C_VEL
LIN {X 0,Y 340.863,Z 398.023,A -85,B 0,C 180,E1 -14209.306,E2 -14209.306} C_VEL
LIN {X 0,Y 341.051,Z 398.003,A -85,B 0,C 180,E1 -14212.898,E2 -14212.898} C_VEL
LIN {X 0,Y 341.162,Z 397.985,A -85,B 0,C 180,E1 -14217.639,E2 -14217.639} C_VEL
LIN {X 0,Y 341.309,Z 397.968,A -85,B 0,C 180,E1 -14220,E2 -14220} C_VEL
LIN {X 0,Y 341.162,Z 397.989,A -85,B 0,C 180,E1 -14222.361,E2 -14222.361} C_VEL
LIN {X 0,Y 341.067,Z 397.998,A -85,B 0,C 180,E1 -14227.102,E2 -14227.102} C_VEL
LIN {X 0,Y 340.863,Z 398.026,A -85,B 0,C 180,E1 -14230.694,E2 -14230.694} C_VEL
LIN {X 0,Y 340.856,Z 398.028,A -85,B 0,C 180,E1 -14234.325,E2 -14234.325} C_VEL
LIN {X 0,Y 340.831,Z 398.032,A -85,B 0,C 180,E1 -14238.467,E2 -14238.467} C_VEL
LIN {X 0,Y 340.747,Z 398.038,A -85,B 0,C 180,E1 -14241.858,E2 -14241.858} C_VEL
LIN {X 0,Y 340.766,Z 398.035,A -85,B 0,C 180,E1 -14245.665,E2 -14245.665} C_VEL
LIN {X 0,Y 340.735,Z 398.044,A -85,B 0,C 180,E1 -14248.32,E2 -14248.32} C_VEL
LIN {X 0,Y 340.698,Z 398.043,A -85,B 0,C 180,E1 -14251.045,E2 -14251.045} C_VEL
LIN {X 0,Y 340.714,Z 398.041,A -85,B 0,C 180,E1 -14255.28,E2 -14255.28} C_VEL
LIN {X 0,Y 340.714,Z 398.045,A -85,B 0,C 180,E1 -14258.389,E2 -14258.389} C_VEL
LIN {X 0,Y 340.726,Z 398.044,A -85,B 0,C 180,E1 -14262.052,E2 -14262.052} C_VEL
LIN {X 0,Y 340.649,Z 398.054,A -85,B 0,C 180,E1 -14266.228,E2 -14266.228} C_VEL
LIN {X 0,Y 340.686,Z 398.047,A -85,B 0,C 180,E1 -14269.754,E2 -14269.754} C_VEL
LIN {X 0,Y 340.704,Z 398.042,A -85,B 0,C 180,E1 -14273.26,E2 -14273.26} C_VEL
LIN {X 0,Y 340.693,Z 398.049,A -85,B 0,C 180,E1 -14276.155,E2 -14276.155} C_VEL
LIN {X 0,Y 340.741,Z 398.04,A -85,B 0,C 180,E1 -14280.33,E2 -14280.33} C_VEL
LIN {X 0,Y 340.804,Z 398.03,A -85,B 0,C 180,E1 -14283.021,E2 -14283.021} C_VEL
LIN {X 0,Y 340.757,Z 398.038,A -85,B 0,C 180,E1 -14285.639,E2 -14285.639} C_VEL
LIN {X 0,Y 340.75,Z 398.038,A -85,B 0,C 180,E1 -14289.475,E2 -14289.475} C_VEL
LIN {X 0,Y 340.86,Z 398.028,A -85,B 0,C 180,E1 -14291.985,E2 -14291.985} C_VEL
LIN {X 0,Y 340.872,Z 398.026,A -85,B 0,C 180,E1 -14295.706,E2 -14295.706} C_VEL
LIN {X 0,Y 340.874,Z 398.022,A -85,B 0,C 180,E1 -14299.307,E2 -14299.307} C_VEL
LIN {X 0,Y 341.079,Z 397.995,A -85,B 0,C 180,E1 -14302.899,E2 -14302.899} C_VEL
LIN {X 0,Y 340.805,Z 398.031,A -85,B 0,C 180,E1 -14305.269,E2 -14305.269} C_VEL
LIN {X 0,Y 341.06,Z 397.998,A -85,B 0,C 180,E1 -14308.82,E2 -14308.82} C_VEL
LIN {X 0,Y 340.151,Z 398.118,A -85,B 0,C 180,E1 -14311.184,E2 -14311.184} C_VEL
LIN {X 0,Y 340.265,Z 401.076,A -85,B 0,C 180,E1 -14314.739,E2 -14314.739} C_VEL
LIN {X 0,Y 340.045,Z 404.282,A -85,B 0,C 180,E1 -14318.319,E2 -14318.319} C_VEL
LIN {X 0,Y 339.852,Z 406.819,A -85,B 0,C 180,E1 -14321.066,E2 -14321.066} C_VEL
LIN {X 0,Y 343.707,Z 420.886,A -85,B 0,C 180,E1 -14321.911,E2 -14321.911} C_VEL
LIN {X 0,Y 346.261,Z 431.812,A -85,B 0,C 180,E1 -14322.737,E2 -14322.737} C_VEL
LIN {X 0,Y 347.113,Z 436.529,A -85,B 0,C 180,E1 -14323.14,E2 -14323.14} C_VEL
LIN {X 0,Y 346.196,Z 447.826,A -85,B 0,C 180,E1 -14324.1,E2 -14324.1} C_VEL
LIN {X 0,Y 345.061,Z 459.332,A -85,B 0,C 180,E1 -14325.354,E2 -14325.354} C_VEL
LIN {X 0,Y 343.88,Z 469.751,A -85,B 0,C 180,E1 -14326.779,E2 -14326.779} C_VEL
LIN {X 0,Y 342.919,Z 478.25,A -85,B 0,C 180,E1 -14328.212,E2 -14328.212} C_VEL
LIN {X 0,Y 341.926,Z 486.093,A -85,B 0,C 180,E1 -14329.825,E2 -14329.825} C_VEL
LIN {X 0,Y 340.972,Z 493.645,A -85,B 0,C 180,E1 -14331.778,E2 -14331.778} C_VEL
LIN {X 0,Y 340.35,Z 499.586,A -85,B 0,C 180,E1 -14333.744,E2 -14333.744} C_VEL
LIN {X 0,Y 339.821,Z 504.164,A -85,B 0,C 180,E1 -14335.741,E2 -14335.741} C_VEL
LIN {X 0,Y 339.586,Z 506.543,A -85,B 0,C 180,E1 -14337.136,E2 -14337.136} C_VEL
LIN {X 0,Y 339.322,Z 508.292,A -85,B 0,C 180,E1 -14338.449,E2 -14338.449} C_VEL
LIN {X 0,Y 339.185,Z 509.52,A -85,B 0,C 180,E1 -14339.82,E2 -14339.82} C_VEL
LIN {X 0,Y 339.133,Z 510.392,A -85,B 0,C 180,E1 -14341.825,E2 -14341.825} C_VEL
LIN {X 0,Y 339.192,Z 510.071,A -85,B 0,C 180,E1 -14344.024,E2 -14344.024} C_VEL
LIN {X 0,Y 339.47,Z 508.44,A -85,B 0,C 180,E1 -14346.156,E2 -14346.156} C_VEL
LIN {X 0,Y 339.939,Z 505.378,A -85,B 0,C 180,E1 -14348.332,E2 -14348.332} C_VEL
LIN {X 0,Y 340.45,Z 501.578,A -85,B 0,C 180,E1 -14350.199,E2 -14350.199} C_VEL
LIN {X 0,Y 341.136,Z 496.375,A -85,B 0,C 180,E1 -14352.126,E2 -14352.126} C_VEL
LIN {X 0,Y 342.129,Z 489.728,A -85,B 0,C 180,E1 -14354.03,E2 -14354.03} C_VEL
LIN {X 0,Y 343.281,Z 481.467,A -85,B 0,C 180,E1 -14355.886,E2 -14355.886} C_VEL
LIN {X 0,Y 344.344,Z 473.797,A -85,B 0,C 180,E1 -14357.285,E2 -14357.285} C_VEL
LIN {X 0,Y 345.582,Z 463.647,A -85,B 0,C 180,E1 -14358.803,E2 -14358.803} C_VEL
LIN {X 0,Y 346.782,Z 452.805,A -85,B 0,C 180,E1 -14360.084,E2 -14360.084} C_VEL
LIN {X 0,Y 347.872,Z 442.082,A -85,B 0,C 180,E1 -14361.089,E2 -14361.089} C_VEL
LIN {X 0,Y 348.083,Z 437.848,A -85,B 0,C 180,E1 -14361.436,E2 -14361.436} C_VEL
LIN {X 0,Y 347.859,Z 436.701,A -85,B 0,C 180,E1 -14361.543,E2 -14361.543} C_VEL
LIN {X 0,Y 346.863,Z 433.435,A -85,B 0,C 180,E1 -14361.869,E2 -14361.869} C_VEL
LIN {X 0,Y 344.421,Z 428.935,A -85,B 0,C 180,E1 -14362.369,E2 -14362.369} C_VEL
LIN {X 0,Y 337.175,Z 418.968,A -85,B 0,C 180,E1 -14363.484,E2 -14363.484} C_VEL
LIN {X 0,Y 334.618,Z 414.152,A -85,B 0,C 180,E1 -14363.894,E2 -14363.894} C_VEL
LIN {X 0,Y 333.982,Z 412.402,A -85,B 0,C 180,E1 -14364.013,E2 -14364.013} C_VEL
LIN {X 0,Y 332.905,Z 409.096,A -85,B 0,C 180,E1 -14364.231,E2 -14364.231} C_VEL
LIN {X 0,Y 333.144,Z 405.869,A -85,B 0,C 180,E1 -14368.17,E2 -14368.17} C_VEL
LIN {X 0,Y 333.381,Z 402.601,A -85,B 0,C 180,E1 -14372.299,E2 -14372.299} C_VEL
LIN {X 0,Y 333.525,Z 400.468,A -85,B 0,C 180,E1 -14375.074,E2 -14375.074} C_VEL
LIN {X 0,Y 333.57,Z 399.48,A -85,B 0,C 180,E1 -14376.402,E2 -14376.402} C_VEL
LIN {X 0,Y 333.599,Z 398.938,A -85,B 0,C 180,E1 -14377.963,E2 -14377.963} C_VEL
LIN {X 0,Y 333.79,Z 398.908,A -85,B 0,C 180,E1 -14381.589,E2 -14381.589} C_VEL
LIN {X 0,Y 333.805,Z 398.906,A -85,B 0,C 180,E1 -14385.576,E2 -14385.576} C_VEL
LIN {X 0,Y 333.83,Z 398.902,A -85,B 0,C 180,E1 -14389.078,E2 -14389.078} C_VEL
LIN {X 0,Y 334.002,Z 398.879,A -85,B 0,C 180,E1 -14392.747,E2 -14392.747} C_VEL
LIN {X 0,Y 333.805,Z 398.903,A -85,B 0,C 180,E1 -14395.169,E2 -14395.169} C_VEL
LIN {X 0,Y 334.102,Z 398.866,A -85,B 0,C 180,E1 -14397.589,E2 -14397.589} C_VEL
LIN {X 0,Y 334.242,Z 398.848,A -85,B 0,C 180,E1 -14400,E2 -14400} C_VEL
LIN {X 0,Y 334.102,Z 398.865,A -85,B 0,C 180,E1 -14402.411,E2 -14402.411} C_VEL
LIN {X 0,Y 334.01,Z 398.88,A -85,B 0,C 180,E1 -14406.039,E2 -14406.039} C_VEL
LIN {X 0,Y 333.954,Z 398.885,A -85,B 0,C 180,E1 -14408.471,E2 -14408.471} C_VEL
LIN {X 0,Y 333.787,Z 398.908,A -85,B 0,C 180,E1 -14412.155,E2 -14412.155} C_VEL
LIN {X 0,Y 333.773,Z 398.906,A -85,B 0,C 180,E1 -14415.886,E2 -14415.886} C_VEL
LIN {X 0,Y 333.793,Z 398.903,A -85,B 0,C 180,E1 -14418.655,E2 -14418.655} C_VEL
LIN {X 0,Y 333.689,Z 398.921,A -85,B 0,C 180,E1 -14422.278,E2 -14422.278} C_VEL
LIN {X 0,Y 333.731,Z 398.912,A -85,B 0,C 180,E1 -14426.247,E2 -14426.247} C_VEL
LIN {X 0,Y 333.686,Z 398.918,A -85,B 0,C 180,E1 -14428.974,E2 -14428.974} C_VEL
LIN {X 0,Y 333.64,Z 398.929,A -85,B 0,C 180,E1 -14432.587,E2 -14432.587} C_VEL
LIN {X 0,Y 333.674,Z 398.928,A -85,B 0,C 180,E1 -14436.139,E2 -14436.139} C_VEL
LIN {X 0,Y 333.671,Z 398.924,A -85,B 0,C 180,E1 -14439.945,E2 -14439.945} C_VEL
LIN {X 0,Y 333.729,Z 399.225,A -85,B 0,C 180,E1 -14440.702,E2 -14440.702} C_VEL
LIN {X 0,Y 334.477,Z 403.572,A -85,B 0,C 180,E1 -14444.406,E2 -14444.406} C_VEL
LIN {X 0,Y 335.327,Z 408.089,A -85,B 0,C 180,E1 -14447.881,E2 -14447.881} C_VEL
LIN {X 0,Y 336.112,Z 412.759,A -85,B 0,C 180,E1 -14451.15,E2 -14451.15} C_VEL
LIN {X 0,Y 336.477,Z 416.364,A -85,B 0,C 180,E1 -14453.468,E2 -14453.468} C_VEL
LIN {X 0,Y 335.835,Z 421.132,A -85,B 0,C 180,E1 -14456.311,E2 -14456.311} C_VEL
LIN {X 0,Y 334.803,Z 428.481,A -85,B 0,C 180,E1 -14460.443,E2 -14460.443} C_VEL
LIN {X 0,Y 333.957,Z 435.828,A -85,B 0,C 180,E1 -14464.383,E2 -14464.383} C_VEL
LIN {X 0,Y 333.353,Z 442.419,A -85,B 0,C 180,E1 -14467.806,E2 -14467.806} C_VEL
LIN {X 0,Y 336.395,Z 457.061,A -85,B 0,C 180,E1 -14468.628,E2 -14468.628} C_VEL
LIN {X 0,Y 338.132,Z 470.482,A -85,B 0,C 180,E1 -14469.575,E2 -14469.575} C_VEL
LIN {X 0,Y 339.056,Z 482.566,A -85,B 0,C 180,E1 -14470.631,E2 -14470.631} C_VEL
LIN {X 0,Y 339.21,Z 487.341,A -85,B 0,C 180,E1 -14471.111,E2 -14471.111} C_VEL
LIN {X 0,Y 337.822,Z 498.196,A -85,B 0,C 180,E1 -14472.287,E2 -14472.287} C_VEL
LIN {X 0,Y 336.448,Z 508.466,A -85,B 0,C 180,E1 -14473.683,E2 -14473.683} C_VEL
LIN {X 0,Y 335.427,Z 517.145,A -85,B 0,C 180,E1 -14475.136,E2 -14475.136} C_VEL
LIN {X 0,Y 334.238,Z 525.963,A -85,B 0,C 180,E1 -14476.936,E2 -14476.936} C_VEL
LIN {X 0,Y 333.32,Z 533.075,A -85,B 0,C 180,E1 -14478.753,E2 -14478.753} C_VEL
LIN {X 0,Y 332.641,Z 539.62,A -85,B 0,C 180,E1 -14480.882,E2 -14480.882} C_VEL
LIN {X 0,Y 332.276,Z 543.952,A -85,B 0,C 180,E1 -14482.709,E2 -14482.709} C_VEL
LIN {X 0,Y 332.181,Z 546.264,A -85,B 0,C 180,E1 -14483.927,E2 -14483.927} C_VEL
LIN {X 0,Y 332.11,Z 548.099,A -85,B 0,C 180,E1 -14485.144,E2 -14485.144} C_VEL
LIN {X 0,Y 332.057,Z 549.497,A -85,B 0,C 180,E1 -14486.359,E2 -14486.359} C_VEL
LIN {X 0,Y 332.133,Z 551.107,A -85,B 0,C 180,E1 -14488.787,E2 -14488.787} C_VEL
LIN {X 0,Y 332.213,Z 551.281,A -85,B 0,C 180,E1 -14490,E2 -14490} C_VEL
LIN {X 0,Y 332.166,Z 551.035,A -85,B 0,C 180,E1 -14491.212,E2 -14491.212} C_VEL
LIN {X 0,Y 332.057,Z 549.36,A -85,B 0,C 180,E1 -14493.64,E2 -14493.64} C_VEL
LIN {X 0,Y 332.115,Z 547.877,A -85,B 0,C 180,E1 -14494.855,E2 -14494.855} C_VEL
LIN {X 0,Y 332.218,Z 544.84,A -85,B 0,C 180,E1 -14496.681,E2 -14496.681} C_VEL
LIN {X 0,Y 332.492,Z 540.734,A -85,B 0,C 180,E1 -14498.508,E2 -14498.508} C_VEL
LIN {X 0,Y 333.116,Z 534.435,A -85,B 0,C 180,E1 -14500.638,E2 -14500.638} C_VEL
LIN {X 0,Y 333.877,Z 527.576,A -85,B 0,C 180,E1 -14502.459,E2 -14502.459} C_VEL
LIN {X 0,Y 334.755,Z 520.586,A -85,B 0,C 180,E1 -14503.971,E2 -14503.971} C_VEL
LIN {X 0,Y 335.966,Z 511.326,A -85,B 0,C 180,E1 -14505.611,E2 -14505.611} C_VEL
LIN {X 0,Y 337.072,Z 500.639,A -85,B 0,C 180,E1 -14507.127,E2 -14507.127} C_VEL
LIN {X 0,Y 338.368,Z 490.184,A -85,B 0,C 180,E1 -14508.309,E2 -14508.309} C_VEL
LIN {X 0,Y 338.856,Z 485.579,A -85,B 0,C 180,E1 -14508.751,E2 -14508.751} C_VEL
LIN {X 0,Y 337.842,Z 473.92,A -85,B 0,C 180,E1 -14509.803,E2 -14509.803} C_VEL
LIN {X 0,Y 336.275,Z 460.905,A -85,B 0,C 180,E1 -14510.725,E2 -14510.725} C_VEL
LIN {X 0,Y 333.972,Z 447.505,A -85,B 0,C 180,E1 -14511.453,E2 -14511.453} C_VEL
LIN {X 0,Y 333.331,Z 443.675,A -85,B 0,C 180,E1 -14511.619,E2 -14511.619} C_VEL
LIN {X 0,Y 334.01,Z 435.9,A -85,B 0,C 180,E1 -14515.629,E2 -14515.629} C_VEL
LIN {X 0,Y 334.807,Z 428.457,A -85,B 0,C 180,E1 -14519.556,E2 -14519.556} C_VEL
LIN {X 0,Y 335.813,Z 420.895,A -85,B 0,C 180,E1 -14523.692,E2 -14523.692} C_VEL
LIN {X 0,Y 336.402,Z 415.855,A -85,B 0,C 180,E1 -14526.541,E2 -14526.541} C_VEL
LIN {X 0,Y 336.063,Z 412.037,A -85,B 0,C 180,E1 -14528.856,E2 -14528.856} C_VEL
LIN {X 0,Y 335.105,Z 406.912,A -85,B 0,C 180,E1 -14532.152,E2 -14532.152} C_VEL
LIN {X 0,Y 334.101,Z 401.228,A -85,B 0,C 180,E1 -14536.039,E2 -14536.039} C_VEL
LIN {X 0,Y 333.688,Z 398.92,A -85,B 0,C 180,E1 -14537.83,E2 -14537.83} C_VEL
LIN {X 0,Y 333.672,Z 398.923,A -85,B 0,C 180,E1 -14541.196,E2 -14541.196} C_VEL
LIN {X 0,Y 333.68,Z 398.92,A -85,B 0,C 180,E1 -14545.225,E2 -14545.225} C_VEL
LIN {X 0,Y 333.624,Z 398.925,A -85,B 0,C 180,E1 -14548.221,E2 -14548.221} C_VEL
LIN {X 0,Y 333.683,Z 398.921,A -85,B 0,C 180,E1 -14551.025,E2 -14551.025} C_VEL
LIN {X 0,Y 333.728,Z 398.911,A -85,B 0,C 180,E1 -14553.753,E2 -14553.753} C_VEL
LIN {X 0,Y 333.713,Z 398.913,A -85,B 0,C 180,E1 -14557.914,E2 -14557.914} C_VEL
LIN {X 0,Y 333.786,Z 398.904,A -85,B 0,C 180,E1 -14561.589,E2 -14561.589} C_VEL
LIN {X 0,Y 333.801,Z 398.902,A -85,B 0,C 180,E1 -14565.576,E2 -14565.576} C_VEL
LIN {X 0,Y 333.826,Z 398.901,A -85,B 0,C 180,E1 -14569.078,E2 -14569.078} C_VEL
LIN {X 0,Y 333.998,Z 398.883,A -85,B 0,C 180,E1 -14572.747,E2 -14572.747} C_VEL
LIN {X 0,Y 333.803,Z 398.903,A -85,B 0,C 180,E1 -14575.169,E2 -14575.169} C_VEL
LIN {X 0,Y 334.099,Z 398.865,A -85,B 0,C 180,E1 -14577.589,E2 -14577.589} C_VEL
LIN {X 0,Y 334.259,Z 398.846,A -85,B 0,C 180,E1 -14580,E2 -14580} C_VEL
LIN {X 0,Y 334.099,Z 398.869,A -85,B 0,C 180,E1 -14582.411,E2 -14582.411} C_VEL
LIN {X 0,Y 334.017,Z 398.876,A -85,B 0,C 180,E1 -14587.253,E2 -14587.253} C_VEL
LIN {X 0,Y 333.826,Z 398.901,A -85,B 0,C 180,E1 -14590.922,E2 -14590.922} C_VEL
LIN {X 0,Y 333.801,Z 398.906,A -85,B 0,C 180,E1 -14594.635,E2 -14594.635} C_VEL
LIN {X 0,Y 333.79,Z 398.907,A -85,B 0,C 180,E1 -14598.656,E2 -14598.656} C_VEL
LIN {X 0,Y 333.686,Z 398.921,A -85,B 0,C 180,E1 -14602.279,E2 -14602.279} C_VEL
LIN {X 0,Y 333.73,Z 398.916,A -85,B 0,C 180,E1 -14606.247,E2 -14606.247} C_VEL
LIN {X 0,Y 333.705,Z 398.915,A -85,B 0,C 180,E1 -14608.973,E2 -14608.973} C_VEL
LIN {X 0,Y 333.638,Z 398.925,A -85,B 0,C 180,E1 -14612.588,E2 -14612.588} C_VEL
LIN {X 0,Y 333.672,Z 398.923,A -85,B 0,C 180,E1 -14616.14,E2 -14616.14} C_VEL
LIN {X 0,Y 333.668,Z 398.918,A -85,B 0,C 180,E1 -14619.19,E2 -14619.19} C_VEL
LIN {X 0,Y 333.657,Z 398.923,A -85,B 0,C 180,E1 -14622.506,E2 -14622.506} C_VEL
LIN {X 0,Y 333.594,Z 398.932,A -85,B 0,C 180,E1 -14625.956,E2 -14625.956} C_VEL
LIN {X 0,Y 333.645,Z 398.921,A -85,B 0,C 180,E1 -14629.316,E2 -14629.316} C_VEL
LIN {X 0,Y 333.664,Z 398.918,A -85,B 0,C 180,E1 -14633.169,E2 -14633.169} C_VEL
LIN {X 0,Y 333.638,Z 398.923,A -85,B 0,C 180,E1 -14636.793,E2 -14636.793} C_VEL
LIN {X 0,Y 333.694,Z 398.918,A -85,B 0,C 180,E1 -14639.714,E2 -14639.714} C_VEL
LIN {X 0,Y 333.74,Z 398.911,A -85,B 0,C 180,E1 -14642.402,E2 -14642.402} C_VEL
LIN {X 0,Y 333.728,Z 398.911,A -85,B 0,C 180,E1 -14645.092,E2 -14645.092} C_VEL
LIN {X 0,Y 333.683,Z 398.917,A -85,B 0,C 180,E1 -14649.02,E2 -14649.02} C_VEL
LIN {X 0,Y 333.796,Z 398.905,A -85,B 0,C 180,E1 -14651.59,E2 -14651.59} C_VEL
LIN {X 0,Y 333.811,Z 398.904,A -85,B 0,C 180,E1 -14655.577,E2 -14655.577} C_VEL
LIN {X 0,Y 333.836,Z 398.898,A -85,B 0,C 180,E1 -14659.079,E2 -14659.079} C_VEL
LIN {X 0,Y 334.029,Z 398.874,A -85,B 0,C 180,E1 -14662.748,E2 -14662.748} C_VEL
LIN {X 0,Y 333.774,Z 398.906,A -85,B 0,C 180,E1 -14665.169,E2 -14665.169} C_VEL
LIN {X 0,Y 334.028,Z 398.874,A -85,B 0,C 180,E1 -14668.795,E2 -14668.795} C_VEL
LIN {X 0,Y 333.097,Z 398.997,A -85,B 0,C 180,E1 -14671.209,E2 -14671.209} C_VEL
LIN {X 0,Y 333.2,Z 402.004,A -85,B 0,C 180,E1 -14674.84,E2 -14674.84} C_VEL
LIN {X 0,Y 332.972,Z 405.316,A -85,B 0,C 180,E1 -14678.497,E2 -14678.497} C_VEL
LIN {X 0,Y 332.796,Z 407.275,A -85,B 0,C 180,E1 -14680.649,E2 -14680.649} C_VEL
LIN {X 0,Y 336.545,Z 420.596,A -85,B 0,C 180,E1 -14681.462,E2 -14681.462} C_VEL
LIN {X 0,Y 339.283,Z 432.314,A -85,B 0,C 180,E1 -14682.365,E2 -14682.365} C_VEL
LIN {X 0,Y 340.247,Z 438.546,A -85,B 0,C 180,E1 -14682.906,E2 -14682.906} C_VEL
LIN {X 0,Y 339.253,Z 450.243,A -85,B 0,C 180,E1 -14683.968,E2 -14683.968} C_VEL
LIN {X 0,Y 338.124,Z 461.088,A -85,B 0,C 180,E1 -14685.213,E2 -14685.213} C_VEL
LIN {X 0,Y 336.912,Z 471.199,A -85,B 0,C 180,E1 -14686.653,E2 -14686.653} C_VEL
LIN {X 0,Y 335.773,Z 480.419,A -85,B 0,C 180,E1 -14688.298,E2 -14688.298} C_VEL
LIN {X 0,Y 334.766,Z 487.94,A -85,B 0,C 180,E1 -14689.947,E2 -14689.947} C_VEL
LIN {X 0,Y 334.005,Z 493.864,A -85,B 0,C 180,E1 -14691.533,E2 -14691.533} C_VEL
LIN {X 0,Y 333.302,Z 500.059,A -85,B 0,C 180,E1 -14693.618,E2 -14693.618} C_VEL
LIN {X 0,Y 332.756,Z 504.624,A -85,B 0,C 180,E1 -14695.656,E2 -14695.656} C_VEL
LIN {X 0,Y 332.388,Z 507.889,A -85,B 0,C 180,E1 -14697.721,E2 -14697.721} C_VEL
LIN {X 0,Y 332.098,Z 509.959,A -85,B 0,C 180,E1 -14699.812,E2 -14699.812} C_VEL
LIN {X 0,Y 332.052,Z 510.88,A -85,B 0,C 180,E1 -14702.154,E2 -14702.154} C_VEL
LIN {X 0,Y 332.127,Z 510.367,A -85,B 0,C 180,E1 -14704.384,E2 -14704.384} C_VEL
LIN {X 0,Y 332.472,Z 508.553,A -85,B 0,C 180,E1 -14706.556,E2 -14706.556} C_VEL
LIN {X 0,Y 332.939,Z 505.567,A -85,B 0,C 180,E1 -14708.644,E2 -14708.644} C_VEL
LIN {X 0,Y 333.557,Z 501.157,A -85,B 0,C 180,E1 -14710.78,E2 -14710.78} C_VEL
LIN {X 0,Y 334.34,Z 496.029,A -85,B 0,C 180,E1 -14712.632,E2 -14712.632} C_VEL
LIN {X 0,Y 335.34,Z 489.217,A -85,B 0,C 180,E1 -14714.555,E2 -14714.555} C_VEL
LIN {X 0,Y 336.626,Z 480.732,A -85,B 0,C 180,E1 -14716.451,E2 -14716.451} C_VEL
LIN {X 0,Y 337.821,Z 472.186,A -85,B 0,C 180,E1 -14717.983,E2 -14717.983} C_VEL
LIN {X 0,Y 339.063,Z 462.491,A -85,B 0,C 180,E1 -14719.389,E2 -14719.389} C_VEL
LIN {X 0,Y 340.205,Z 452.532,A -85,B 0,C 180,E1 -14720.561,E2 -14720.561} C_VEL
LIN {X 0,Y 341.351,Z 441.438,A -85,B 0,C 180,E1 -14721.602,E2 -14721.602} C_VEL
LIN {X 0,Y 341.293,Z 438.653,A -85,B 0,C 180,E1 -14721.846,E2 -14721.846} C_VEL
LIN {X 0,Y 338.919,Z 428.203,A -85,B 0,C 180,E1 -14722.8,E2 -14722.8} C_VEL
LIN {X 0,Y 334.997,Z 415.37,A -85,B 0,C 180,E1 -14723.809,E2 -14723.809} C_VEL
LIN {X 0,Y 333.982,Z 412.402,A -85,B 0,C 180,E1 -14724.013,E2 -14724.013} C_VEL
LIN {X 0,Y 332.926,Z 410.229,A -85,B 0,C 180,E1 -14724.305,E2 -14724.305} C_VEL
LIN {X 0,Y 331.371,Z 408.768,A -85,B 0,C 180,E1 -14724.876,E2 -14724.876} C_VEL
LIN {X 0,Y 328.821,Z 408.11,A -85,B 0,C 180,E1 -14726.129,E2 -14726.129} C_VEL
LIN {X 0,Y 326.852,Z 407.296,A -85,B 0,C 180,E1 -14727.647,E2 -14727.647} C_VEL
LIN {X 0,Y 326.145,Z 406.051,A -85,B 0,C 180,E1 -14729.194,E2 -14729.194} C_VEL
LIN {X 0,Y 326.371,Z 403.037,A -85,B 0,C 180,E1 -14733.114,E2 -14733.114} C_VEL
LIN {X 0,Y 326.543,Z 400.994,A -85,B 0,C 180,E1 -14735.862,E2 -14735.862} C_VEL
LIN {X 0,Y 326.545,Z 399.817,A -85,B 0,C 180,E1 -14737.736,E2 -14737.736} C_VEL
LIN {X 0,Y 326.741,Z 399.787,A -85,B 0,C 180,E1 -14741.177,E2 -14741.177} C_VEL
LIN {X 0,Y 326.759,Z 399.784,A -85,B 0,C 180,E1 -14745.433,E2 -14745.433} C_VEL
LIN {X 0,Y 326.766,Z 399.781,A -85,B 0,C 180,E1 -14748.839,E2 -14748.839} C_VEL
LIN {X 0,Y 326.954,Z 399.757,A -85,B 0,C 180,E1 -14752.59,E2 -14752.59} C_VEL
LIN {X 0,Y 326.772,Z 399.779,A -85,B 0,C 180,E1 -14755.065,E2 -14755.065} C_VEL
LIN {X 0,Y 327.043,Z 399.745,A -85,B 0,C 180,E1 -14757.537,E2 -14757.537} C_VEL
LIN {X 0,Y 327.193,Z 399.726,A -85,B 0,C 180,E1 -14760,E2 -14760} C_VEL
LIN {X 0,Y 327.043,Z 399.745,A -85,B 0,C 180,E1 -14762.463,E2 -14762.463} C_VEL
LIN {X 0,Y 326.985,Z 399.755,A -85,B 0,C 180,E1 -14766.169,E2 -14766.169} C_VEL
LIN {X 0,Y 326.802,Z 399.777,A -85,B 0,C 180,E1 -14769.907,E2 -14769.907} C_VEL
LIN {X 0,Y 326.755,Z 399.78,A -85,B 0,C 180,E1 -14773.685,E2 -14773.685} C_VEL
LIN {X 0,Y 326.695,Z 399.792,A -85,B 0,C 180,E1 -14777.528,E2 -14777.528} C_VEL
LIN {X 0,Y 326.664,Z 399.796,A -85,B 0,C 180,E1 -14780.135,E2 -14780.135} C_VEL
LIN {X 0,Y 326.648,Z 399.798,A -85,B 0,C 180,E1 -14784.129,E2 -14784.129} C_VEL
LIN {X 0,Y 326.679,Z 399.791,A -85,B 0,C 180,E1 -14786.858,E2 -14786.858} C_VEL
LIN {X 0,Y 326.631,Z 399.8,A -85,B 0,C 180,E1 -14790.61,E2 -14790.61} C_VEL
LIN {X 0,Y 326.604,Z 399.808,A -85,B 0,C 180,E1 -14794.02,E2 -14794.02} C_VEL
LIN {X 0,Y 326.627,Z 399.802,A -85,B 0,C 180,E1 -14797.239,E2 -14797.239} C_VEL
LIN {X 0,Y 326.653,Z 400.002,A -85,B 0,C 180,E1 -14799.93,E2 -14799.93} C_VEL
LIN {X 0,Y 327.326,Z 403.863,A -85,B 0,C 180,E1 -14803.399,E2 -14803.399} C_VEL
LIN {X 0,Y 328.08,Z 408.007,A -85,B 0,C 180,E1 -14806.747,E2 -14806.747} C_VEL
LIN {X 0,Y 328.935,Z 412.816,A -85,B 0,C 180,E1 -14810.28,E2 -14810.28} C_VEL
LIN {X 0,Y 329.377,Z 415.52,A -85,B 0,C 180,E1 -14812.137,E2 -14812.137} C_VEL
LIN {X 0,Y 329.373,Z 418.698,A -85,B 0,C 180,E1 -14814.177,E2 -14814.177} C_VEL
LIN {X 0,Y 328.407,Z 424.538,A -85,B 0,C 180,E1 -14817.656,E2 -14817.656} C_VEL
LIN {X 0,Y 327.589,Z 430.595,A -85,B 0,C 180,E1 -14821.105,E2 -14821.105} C_VEL
LIN {X 0,Y 326.832,Z 436.935,A -85,B 0,C 180,E1 -14824.575,E2 -14824.575} C_VEL
LIN {X 0,Y 326.364,Z 442.037,A -85,B 0,C 180,E1 -14827.258,E2 -14827.258} C_VEL
LIN {X 0,Y 329.378,Z 455.938,A -85,B 0,C 180,E1 -14828.063,E2 -14828.063} C_VEL
LIN {X 0,Y 331.078,Z 468.029,A -85,B 0,C 180,E1 -14828.932,E2 -14828.932} C_VEL
LIN {X 0,Y 332.058,Z 480.576,A -85,B 0,C 180,E1 -14830.025,E2 -14830.025} C_VEL
LIN {X 0,Y 332.327,Z 488.733,A -85,B 0,C 180,E1 -14830.865,E2 -14830.865} C_VEL
LIN {X 0,Y 330.707,Z 500.381,A -85,B 0,C 180,E1 -14832.212,E2 -14832.212} C_VEL
LIN {X 0,Y 329.417,Z 509.822,A -85,B 0,C 180,E1 -14833.58,E2 -14833.58} C_VEL
LIN {X 0,Y 328.301,Z 518.485,A -85,B 0,C 180,E1 -14835.115,E2 -14835.115} C_VEL
LIN {X 0,Y 327.117,Z 526.93,A -85,B 0,C 180,E1 -14836.962,E2 -14836.962} C_VEL
LIN {X 0,Y 326.188,Z 533.764,A -85,B 0,C 180,E1 -14838.819,E2 -14838.819} C_VEL
LIN {X 0,Y 325.605,Z 539.256,A -85,B 0,C 180,E1 -14840.684,E2 -14840.684} C_VEL
LIN {X 0,Y 325.205,Z 543.568,A -85,B 0,C 180,E1 -14842.55,E2 -14842.55} C_VEL
LIN {X 0,Y 325.102,Z 546.119,A -85,B 0,C 180,E1 -14843.946,E2 -14843.946} C_VEL
LIN {X 0,Y 324.985,Z 549.088,A -85,B 0,C 180,E1 -14846.28,E2 -14846.28} C_VEL
LIN {X 0,Y 325.039,Z 550.684,A -85,B 0,C 180,E1 -14848.761,E2 -14848.761} C_VEL
LIN {X 0,Y 325.137,Z 550.846,A -85,B 0,C 180,E1 -14850,E2 -14850} C_VEL
LIN {X 0,Y 325.072,Z 550.593,A -85,B 0,C 180,E1 -14851.238,E2 -14851.238} C_VEL
LIN {X 0,Y 324.986,Z 548.903,A -85,B 0,C 180,E1 -14853.719,E2 -14853.719} C_VEL
LIN {X 0,Y 325.083,Z 545.783,A -85,B 0,C 180,E1 -14856.022,E2 -14856.022} C_VEL
LIN {X 0,Y 325.301,Z 541.706,A -85,B 0,C 180,E1 -14858.072,E2 -14858.072} C_VEL
LIN {X 0,Y 325.802,Z 536.819,A -85,B 0,C 180,E1 -14859.937,E2 -14859.937} C_VEL
LIN {X 0,Y 326.415,Z 530.648,A -85,B 0,C 180,E1 -14861.802,E2 -14861.802} C_VEL
LIN {X 0,Y 327.476,Z 522.992,A -85,B 0,C 180,E1 -14863.654,E2 -14863.654} C_VEL
LIN {X 0,Y 328.68,Z 513.851,A -85,B 0,C 180,E1 -14865.416,E2 -14865.416} C_VEL
LIN {X 0,Y 329.818,Z 503.431,A -85,B 0,C 180,E1 -14867.037,E2 -14867.037} C_VEL
LIN {X 0,Y 331.235,Z 492.317,A -85,B 0,C 180,E1 -14868.397,E2 -14868.397} C_VEL
LIN {X 0,Y 331.936,Z 486.417,A -85,B 0,C 180,E1 -14868.997,E2 -14868.997} C_VEL
LIN {X 0,Y 330.949,Z 474.399,A -85,B 0,C 180,E1 -14870.124,E2 -14870.124} C_VEL
LIN {X 0,Y 329.455,Z 461.73,A -85,B 0,C 180,E1 -14871.066,E2 -14871.066} C_VEL
LIN {X 0,Y 327.208,Z 448.312,A -85,B 0,C 180,E1 -14871.829,E2 -14871.829} C_VEL
LIN {X 0,Y 326.306,Z 443.27,A -85,B 0,C 180,E1 -14872.075,E2 -14872.075} C_VEL
LIN {X 0,Y 327.035,Z 435.598,A -85,B 0,C 180,E1 -14876.138,E2 -14876.138} C_VEL
LIN {X 0,Y 327.91,Z 428.052,A -85,B 0,C 180,E1 -14880.242,E2 -14880.242} C_VEL
LIN {X 0,Y 328.783,Z 421.744,A -85,B 0,C 180,E1 -14883.763,E2 -14883.763} C_VEL
LIN {X 0,Y 329.403,Z 416.722,A -85,B 0,C 180,E1 -14886.682,E2 -14886.682} C_VEL
LIN {X 0,Y 329.029,Z 413.045,A -85,B 0,C 180,E1 -14888.964,E2 -14888.964} C_VEL
LIN {X 0,Y 328.069,Z 407.803,A -85,B 0,C 180,E1 -14892.399,E2 -14892.399} C_VEL
LIN {X 0,Y 327.212,Z 402.881,A -85,B 0,C 180,E1 -14895.838,E2 -14895.838} C_VEL
LIN {X 0,Y 326.646,Z 399.798,A -85,B 0,C 180,E1 -14898.165,E2 -14898.165} C_VEL
LIN {X 0,Y 326.638,Z 399.799,A -85,B 0,C 180,E1 -14901.393,E2 -14901.393} C_VEL
LIN {X 0,Y 326.614,Z 399.802,A -85,B 0,C 180,E1 -14904.85,E2 -14904.85} C_VEL
LIN {X 0,Y 326.602,Z 399.801,A -85,B 0,C 180,E1 -14907.455,E2 -14907.455} C_VEL
LIN {X 0,Y 326.641,Z 399.795,A -85,B 0,C 180,E1 -14910.339,E2 -14910.339} C_VEL
LIN {X 0,Y 326.683,Z 399.791,A -85,B 0,C 180,E1 -14914.516,E2 -14914.516} C_VEL
LIN {X 0,Y 326.641,Z 399.797,A -85,B 0,C 180,E1 -14918.545,E2 -14918.545} C_VEL
LIN {X 0,Y 326.738,Z 399.784,A -85,B 0,C 180,E1 -14921.177,E2 -14921.177} C_VEL
LIN {X 0,Y 326.756,Z 399.78,A -85,B 0,C 180,E1 -14925.433,E2 -14925.433} C_VEL
LIN {X 0,Y 326.762,Z 399.784,A -85,B 0,C 180,E1 -14928.839,E2 -14928.839} C_VEL
LIN {X 0,Y 326.951,Z 399.76,A -85,B 0,C 180,E1 -14932.59,E2 -14932.59} C_VEL
LIN {X 0,Y 326.769,Z 399.78,A -85,B 0,C 180,E1 -14935.065,E2 -14935.065} C_VEL
LIN {X 0,Y 327.04,Z 399.744,A -85,B 0,C 180,E1 -14937.537,E2 -14937.537} C_VEL
LIN {X 0,Y 327.21,Z 399.724,A -85,B 0,C 180,E1 -14940,E2 -14940} C_VEL
LIN {X 0,Y 327.04,Z 399.749,A -85,B 0,C 180,E1 -14942.463,E2 -14942.463} C_VEL
LIN {X 0,Y 326.963,Z 399.753,A -85,B 0,C 180,E1 -14946.658,E2 -14946.658} C_VEL
LIN {X 0,Y 326.806,Z 399.774,A -85,B 0,C 180,E1 -14949.907,E2 -14949.907} C_VEL
LIN {X 0,Y 326.752,Z 399.78,A -85,B 0,C 180,E1 -14953.686,E2 -14953.686} C_VEL
LIN {X 0,Y 326.692,Z 399.788,A -85,B 0,C 180,E1 -14957.529,E2 -14957.529} C_VEL
LIN {X 0,Y 326.658,Z 399.795,A -85,B 0,C 180,E1 -14960.135,E2 -14960.135} C_VEL
LIN {X 0,Y 326.645,Z 399.796,A -85,B 0,C 180,E1 -14964.13,E2 -14964.13} C_VEL
LIN {X 0,Y 326.679,Z 399.791,A -85,B 0,C 180,E1 -14966.858,E2 -14966.858} C_VEL
LIN {X 0,Y 326.633,Z 399.797,A -85,B 0,C 180,E1 -14970.612,E2 -14970.612} C_VEL
LIN {X 0,Y 326.602,Z 399.802,A -85,B 0,C 180,E1 -14974.02,E2 -14974.02} C_VEL
LIN {X 0,Y 326.625,Z 399.796,A -85,B 0,C 180,E1 -14977.24,E2 -14977.24} C_VEL
LIN {X 0,Y 326.6,Z 399.804,A -85,B 0,C 180,E1 -14980.208,E2 -14980.208} C_VEL
LIN {X 0,Y 326.568,Z 399.804,A -85,B 0,C 180,E1 -14983.525,E2 -14983.525} C_VEL
LIN {X 0,Y 326.573,Z 399.802,A -85,B 0,C 180,E1 -14987.029,E2 -14987.029} C_VEL
LIN {X 0,Y 326.61,Z 399.797,A -85,B 0,C 180,E1 -14990.774,E2 -14990.774} C_VEL
LIN {X 0,Y 326.612,Z 399.799,A -85,B 0,C 180,E1 -14994.481,E2 -14994.481} C_VEL
LIN {X 0,Y 326.609,Z 399.799,A -85,B 0,C 180,E1 -14997.457,E2 -14997.457} C_VEL
LIN {X 0,Y 326.648,Z 399.796,A -85,B 0,C 180,E1 -15000.341,E2 -15000.341} C_VEL
LIN {X 0,Y 326.691,Z 399.788,A -85,B 0,C 180,E1 -15004.517,E2 -15004.517} C_VEL
LIN {X 0,Y 326.648,Z 399.794,A -85,B 0,C 180,E1 -15008.546,E2 -15008.546} C_VEL
LIN {X 0,Y 326.746,Z 399.781,A -85,B 0,C 180,E1 -15011.178,E2 -15011.178} C_VEL
LIN {X 0,Y 326.765,Z 399.78,A -85,B 0,C 180,E1 -15015.434,E2 -15015.434} C_VEL
LIN {X 0,Y 326.773,Z 399.777,A -85,B 0,C 180,E1 -15018.84,E2 -15018.84} C_VEL
LIN {X 0,Y 326.983,Z 399.752,A -85,B 0,C 180,E1 -15022.591,E2 -15022.591} C_VEL
LIN {X 0,Y 326.999,Z 399.755,A -85,B 0,C 180,E1 -15023.831,E2 -15023.831} C_VEL
LIN {X 0,Y 326.996,Z 399.75,A -85,B 0,C 180,E1 -15028.769,E2 -15028.769} C_VEL
LIN {X 0,Y 326.043,Z 399.875,A -85,B 0,C 180,E1 -15031.235,E2 -15031.235} C_VEL
LIN {X 0,Y 326.139,Z 402.931,A -85,B 0,C 180,E1 -15034.945,E2 -15034.945} C_VEL
LIN {X 0,Y 325.886,Z 406.298,A -85,B 0,C 180,E1 -15038.683,E2 -15038.683} C_VEL
LIN {X 0,Y 325.793,Z 407.743,A -85,B 0,C 180,E1 -15040.213,E2 -15040.213} C_VEL
LIN {X 0,Y 329.38,Z 420.226,A -85,B 0,C 180,E1 -15040.995,E2 -15040.995} C_VEL
LIN {X 0,Y 332.145,Z 431.932,A -85,B 0,C 180,E1 -15041.906,E2 -15041.906} C_VEL
LIN {X 0,Y 333.456,Z 439.512,A -85,B 0,C 180,E1 -15042.584,E2 -15042.584} C_VEL
LIN {X 0,Y 332.401,Z 451.394,A -85,B 0,C 180,E1 -15043.701,E2 -15043.701} C_VEL
LIN {X 0,Y 331.14,Z 462.876,A -85,B 0,C 180,E1 -15045.069,E2 -15045.069} C_VEL
LIN {X 0,Y 329.902,Z 472.649,A -85,B 0,C 180,E1 -15046.533,E2 -15046.533} C_VEL
LIN {X 0,Y 328.834,Z 480.915,A -85,B 0,C 180,E1 -15048.053,E2 -15048.053} C_VEL
LIN {X 0,Y 327.806,Z 488.318,A -85,B 0,C 180,E1 -15049.709,E2 -15049.709} C_VEL
LIN {X 0,Y 326.964,Z 494.596,A -85,B 0,C 180,E1 -15051.433,E2 -15051.433} C_VEL
LIN {X 0,Y 326.268,Z 500.528,A -85,B 0,C 180,E1 -15053.484,E2 -15053.484} C_VEL
LIN {X 0,Y 325.71,Z 505.079,A -85,B 0,C 180,E1 -15055.566,E2 -15055.566} C_VEL
LIN {X 0,Y 325.312,Z 508.314,A -85,B 0,C 180,E1 -15057.654,E2 -15057.654} C_VEL
LIN {X 0,Y 325.005,Z 510.613,A -85,B 0,C 180,E1 -15060.12,E2 -15060.12} C_VEL
LIN {X 0,Y 324.978,Z 511.321,A -85,B 0,C 180,E1 -15062.497,E2 -15062.497} C_VEL
LIN {X 0,Y 325.111,Z 510.623,A -85,B 0,C 180,E1 -15064.769,E2 -15064.769} C_VEL
LIN {X 0,Y 325.526,Z 508.427,A -85,B 0,C 180,E1 -15067.193,E2 -15067.193} C_VEL
LIN {X 0,Y 326.14,Z 504.56,A -85,B 0,C 180,E1 -15069.62,E2 -15069.62} C_VEL
LIN {X 0,Y 326.902,Z 499.605,A -85,B 0,C 180,E1 -15071.794,E2 -15071.794} C_VEL
LIN {X 0,Y 327.834,Z 493.764,A -85,B 0,C 180,E1 -15073.738,E2 -15073.738} C_VEL
LIN {X 0,Y 329.036,Z 486.038,A -85,B 0,C 180,E1 -15075.74,E2 -15075.74} C_VEL
LIN {X 0,Y 330.359,Z 477.61,A -85,B 0,C 180,E1 -15077.481,E2 -15077.481} C_VEL
LIN {X 0,Y 331.57,Z 469.04,A -85,B 0,C 180,E1 -15078.922,E2 -15078.922} C_VEL
LIN {X 0,Y 332.799,Z 459.845,A -85,B 0,C 180,E1 -15080.188,E2 -15080.188} C_VEL
LIN {X 0,Y 333.964,Z 449.434,A -85,B 0,C 180,E1 -15081.352,E2 -15081.352} C_VEL
LIN {X 0,Y 334.794,Z 441.072,A -85,B 0,C 180,E1 -15082.119,E2 -15082.119} C_VEL
LIN {X 0,Y 332.615,Z 430.875,A -85,B 0,C 180,E1 -15083.107,E2 -15083.107} C_VEL
LIN {X 0,Y 328.767,Z 417.987,A -85,B 0,C 180,E1 -15084.183,E2 -15084.183} C_VEL
LIN {X 0,Y 325.911,Z 409.565,A -85,B 0,C 180,E1 -15084.804,E2 -15084.804} C_VEL
LIN {X 0,Y 326.091,Z 407.47,A -85,B 0,C 180,E1 -15087.397,E2 -15087.397} C_VEL
LIN {X 0,Y 326.145,Z 406.051,A -85,B 0,C 180,E1 -15089.194,E2 -15089.194} C_VEL
LIN {X 0,Y 325.556,Z 405.358,A -85,B 0,C 180,E1 -15090.218,E2 -15090.218} C_VEL
LIN {X 0,Y 322.833,Z 404.505,A -85,B 0,C 180,E1 -15091.895,E2 -15091.895} C_VEL
LIN {X 0,Y 320.504,Z 403.859,A -85,B 0,C 180,E1 -15093.254,E2 -15093.254} C_VEL
LIN {X 0,Y 319.515,Z 403.247,A -85,B 0,C 180,E1 -15094.301,E2 -15094.301} C_VEL
LIN {X 0,Y 319.441,Z 403.001,A -85,B 0,C 180,E1 -15094.655,E2 -15094.655} C_VEL
LIN {X 0,Y 319.506,Z 400.694,A -85,B 0,C 180,E1 -15098.041,E2 -15098.041} C_VEL
LIN {X 0,Y 319.685,Z 400.666,A -85,B 0,C 180,E1 -15100.962,E2 -15100.962} C_VEL
LIN {X 0,Y 319.727,Z 400.66,A -85,B 0,C 180,E1 -15105.276,E2 -15105.276} C_VEL
LIN {X 0,Y 319.748,Z 400.657,A -85,B 0,C 180,E1 -15109.872,E2 -15109.872} C_VEL
LIN {X 0,Y 319.909,Z 400.634,A -85,B 0,C 180,E1 -15112.425,E2 -15112.425} C_VEL
LIN {X 0,Y 319.741,Z 400.654,A -85,B 0,C 180,E1 -15114.956,E2 -15114.956} C_VEL
LIN {X 0,Y 319.987,Z 400.624,A -85,B 0,C 180,E1 -15117.482,E2 -15117.482} C_VEL
LIN {X 0,Y 320.145,Z 400.603,A -85,B 0,C 180,E1 -15120,E2 -15120} C_VEL
LIN {X 0,Y 319.987,Z 400.623,A -85,B 0,C 180,E1 -15122.518,E2 -15122.518} C_VEL
LIN {X 0,Y 319.939,Z 400.634,A -85,B 0,C 180,E1 -15126.306,E2 -15126.306} C_VEL
LIN {X 0,Y 319.833,Z 400.646,A -85,B 0,C 180,E1 -15128.848,E2 -15128.848} C_VEL
LIN {X 0,Y 319.678,Z 400.663,A -85,B 0,C 180,E1 -15132.7,E2 -15132.7} C_VEL
LIN {X 0,Y 319.695,Z 400.662,A -85,B 0,C 180,E1 -15135.296,E2 -15135.296} C_VEL
LIN {X 0,Y 319.672,Z 400.662,A -85,B 0,C 180,E1 -15139.255,E2 -15139.255} C_VEL
LIN {X 0,Y 319.567,Z 400.68,A -85,B 0,C 180,E1 -15143.32,E2 -15143.32} C_VEL
LIN {X 0,Y 319.615,Z 400.671,A -85,B 0,C 180,E1 -15146.09,E2 -15146.09} C_VEL
LIN {X 0,Y 319.576,Z 400.675,A -85,B 0,C 180,E1 -15148.935,E2 -15148.935} C_VEL
LIN {X 0,Y 319.527,Z 400.687,A -85,B 0,C 180,E1 -15151.862,E2 -15151.862} C_VEL
LIN {X 0,Y 319.577,Z 400.681,A -85,B 0,C 180,E1 -15155.543,E2 -15155.543} C_VEL
LIN {X 0,Y 319.624,Z 400.859,A -85,B 0,C 180,E1 -15159.21,E2 -15159.21} C_VEL
LIN {X 0,Y 320.269,Z 404.777,A -85,B 0,C 180,E1 -15162.864,E2 -15162.864} C_VEL
LIN {X 0,Y 321.014,Z 408.825,A -85,B 0,C 180,E1 -15166.259,E2 -15166.259} C_VEL
LIN {X 0,Y 321.724,Z 412.445,A -85,B 0,C 180,E1 -15169.055,E2 -15169.055} C_VEL
LIN {X 0,Y 322.396,Z 417.163,A -85,B 0,C 180,E1 -15172.384,E2 -15172.384} C_VEL
LIN {X 0,Y 322.384,Z 419.52,A -85,B 0,C 180,E1 -15173.943,E2 -15173.943} C_VEL
LIN {X 0,Y 321.566,Z 424.305,A -85,B 0,C 180,E1 -15176.881,E2 -15176.881} C_VEL
LIN {X 0,Y 320.691,Z 430.367,A -85,B 0,C 180,E1 -15180.456,E2 -15180.456} C_VEL
LIN {X 0,Y 319.825,Z 437.147,A -85,B 0,C 180,E1 -15184.284,E2 -15184.284} C_VEL
LIN {X 0,Y 319.374,Z 441.5,A -85,B 0,C 180,E1 -15186.666,E2 -15186.666} C_VEL
LIN {X 0,Y 322.499,Z 455.604,A -85,B 0,C 180,E1 -15187.519,E2 -15187.519} C_VEL
LIN {X 0,Y 324.195,Z 467.148,A -85,B 0,C 180,E1 -15188.375,E2 -15188.375} C_VEL
LIN {X 0,Y 325.166,Z 478.925,A -85,B 0,C 180,E1 -15189.422,E2 -15189.422} C_VEL
LIN {X 0,Y 325.582,Z 488.64,A -85,B 0,C 180,E1 -15190.453,E2 -15190.453} C_VEL
LIN {X 0,Y 323.94,Z 500.216,A -85,B 0,C 180,E1 -15191.828,E2 -15191.828} C_VEL
LIN {X 0,Y 322.578,Z 509.609,A -85,B 0,C 180,E1 -15193.221,E2 -15193.221} C_VEL
LIN {X 0,Y 321.429,Z 518.224,A -85,B 0,C 180,E1 -15194.789,E2 -15194.789} C_VEL
LIN {X 0,Y 320.161,Z 526.632,A -85,B 0,C 180,E1 -15196.674,E2 -15196.674} C_VEL
LIN {X 0,Y 319.165,Z 533.441,A -85,B 0,C 180,E1 -15198.569,E2 -15198.569} C_VEL
LIN {X 0,Y 318.568,Z 538.912,A -85,B 0,C 180,E1 -15200.476,E2 -15200.476} C_VEL
LIN {X 0,Y 318.139,Z 543.202,A -85,B 0,C 180,E1 -15202.383,E2 -15202.383} C_VEL
LIN {X 0,Y 318.009,Z 545.993,A -85,B 0,C 180,E1 -15203.99,E2 -15203.99} C_VEL
LIN {X 0,Y 317.914,Z 548.684,A -85,B 0,C 180,E1 -15206.197,E2 -15206.197} C_VEL
LIN {X 0,Y 317.945,Z 550.26,A -85,B 0,C 180,E1 -15208.733,E2 -15208.733} C_VEL
LIN {X 0,Y 318.064,Z 550.412,A -85,B 0,C 180,E1 -15210,E2 -15210} C_VEL
LIN {X 0,Y 317.979,Z 550.15,A -85,B 0,C 180,E1 -15211.266,E2 -15211.266} C_VEL
LIN {X 0,Y 317.916,Z 548.443,A -85,B 0,C 180,E1 -15213.802,E2 -15213.802} C_VEL
LIN {X 0,Y 318.005,Z 545.558,A -85,B 0,C 180,E1 -15216.004,E2 -15216.004} C_VEL
LIN {X 0,Y 318.241,Z 541.201,A -85,B 0,C 180,E1 -15218.253,E2 -15218.253} C_VEL
LIN {X 0,Y 318.755,Z 536.29,A -85,B 0,C 180,E1 -15220.159,E2 -15220.159} C_VEL
LIN {X 0,Y 319.404,Z 530.091,A -85,B 0,C 180,E1 -15222.065,E2 -15222.065} C_VEL
LIN {X 0,Y 320.516,Z 522.395,A -85,B 0,C 180,E1 -15223.957,E2 -15223.957} C_VEL
LIN {X 0,Y 321.733,Z 513.617,A -85,B 0,C 180,E1 -15225.683,E2 -15225.683} C_VEL
LIN {X 0,Y 322.842,Z 503.806,A -85,B 0,C 180,E1 -15227.253,E2 -15227.253} C_VEL
LIN {X 0,Y 324.291,Z 492.94,A -85,B 0,C 180,E1 -15228.642,E2 -15228.642} C_VEL
LIN {X 0,Y 325.01,Z 487.159,A -85,B 0,C 180,E1 -15229.254,E2 -15229.254} C_VEL
LIN {X 0,Y 324.053,Z 474.811,A -85,B 0,C 180,E1 -15230.456,E2 -15230.456} C_VEL
LIN {X 0,Y 322.589,Z 462.174,A -85,B 0,C 180,E1 -15231.44,E2 -15231.44} C_VEL
LIN {X 0,Y 320.402,Z 448.903,A -85,B 0,C 180,E1 -15232.233,E2 -15232.233} C_VEL
LIN {X 0,Y 319.279,Z 442.876,A -85,B 0,C 180,E1 -15232.53,E2 -15232.53} C_VEL
LIN {X 0,Y 320.077,Z 435.132,A -85,B 0,C 180,E1 -15236.751,E2 -15236.751} C_VEL
LIN {X 0,Y 320.839,Z 428.841,A -85,B 0,C 180,E1 -15240.252,E2 -15240.252} C_VEL
LIN {X 0,Y 321.782,Z 422.492,A -85,B 0,C 180,E1 -15243.906,E2 -15243.906} C_VEL
LIN {X 0,Y 322.358,Z 417.512,A -85,B 0,C 180,E1 -15246.854,E2 -15246.854} C_VEL
LIN {X 0,Y 321.936,Z 413.73,A -85,B 0,C 180,E1 -15249.277,E2 -15249.277} C_VEL
LIN {X 0,Y 320.994,Z 408.599,A -85,B 0,C 180,E1 -15252.743,E2 -15252.743} C_VEL
LIN {X 0,Y 320.116,Z 403.466,A -85,B 0,C 180,E1 -15256.426,E2 -15256.426} C_VEL
LIN {X 0,Y 319.57,Z 400.679,A -85,B 0,C 180,E1 -15258.604,E2 -15258.604} C_VEL
LIN {X 0,Y 319.577,Z 400.678,A -85,B 0,C 180,E1 -15262.342,E2 -15262.342} C_VEL
LIN {X 0,Y 319.555,Z 400.681,A -85,B 0,C 180,E1 -15265.123,E2 -15265.123} C_VEL
LIN {X 0,Y 319.56,Z 400.681,A -85,B 0,C 180,E1 -15269.059,E2 -15269.059} C_VEL
LIN {X 0,Y 319.599,Z 400.674,A -85,B 0,C 180,E1 -15272.497,E2 -15272.497} C_VEL
LIN {X 0,Y 319.598,Z 400.673,A -85,B 0,C 180,E1 -15275.303,E2 -15275.303} C_VEL
LIN {X 0,Y 319.591,Z 400.673,A -85,B 0,C 180,E1 -15278.047,E2 -15278.047} C_VEL
LIN {X 0,Y 319.682,Z 400.665,A -85,B 0,C 180,E1 -15280.962,E2 -15280.962} C_VEL
LIN {X 0,Y 319.724,Z 400.657,A -85,B 0,C 180,E1 -15285.276,E2 -15285.276} C_VEL
LIN {X 0,Y 319.745,Z 400.653,A -85,B 0,C 180,E1 -15289.873,E2 -15289.873} C_VEL
LIN {X 0,Y 319.905,Z 400.636,A -85,B 0,C 180,E1 -15292.426,E2 -15292.426} C_VEL
LIN {X 0,Y 319.739,Z 400.656,A -85,B 0,C 180,E1 -15294.956,E2 -15294.956} C_VEL
LIN {X 0,Y 319.984,Z 400.623,A -85,B 0,C 180,E1 -15297.482,E2 -15297.482} C_VEL
LIN {X 0,Y 320.162,Z 400.602,A -85,B 0,C 180,E1 -15300,E2 -15300} C_VEL
LIN {X 0,Y 319.984,Z 400.628,A -85,B 0,C 180,E1 -15302.518,E2 -15302.518} C_VEL
LIN {X 0,Y 319.923,Z 400.631,A -85,B 0,C 180,E1 -15306.649,E2 -15306.649} C_VEL
LIN {X 0,Y 319.75,Z 400.654,A -85,B 0,C 180,E1 -15310.128,E2 -15310.128} C_VEL
LIN {X 0,Y 319.724,Z 400.658,A -85,B 0,C 180,E1 -15314.725,E2 -15314.725} C_VEL
LIN {X 0,Y 319.683,Z 400.661,A -85,B 0,C 180,E1 -15319.038,E2 -15319.038} C_VEL
LIN {X 0,Y 319.564,Z 400.674,A -85,B 0,C 180,E1 -15323.32,E2 -15323.32} C_VEL
LIN {X 0,Y 319.629,Z 400.67,A -85,B 0,C 180,E1 -15326.089,E2 -15326.089} C_VEL
LIN {X 0,Y 319.584,Z 400.674,A -85,B 0,C 180,E1 -15328.934,E2 -15328.934} C_VEL
LIN {X 0,Y 319.527,Z 400.681,A -85,B 0,C 180,E1 -15331.863,E2 -15331.863} C_VEL
LIN {X 0,Y 319.575,Z 400.674,A -85,B 0,C 180,E1 -15335.544,E2 -15335.544} C_VEL
LIN {X 0,Y 319.594,Z 400.675,A -85,B 0,C 180,E1 -15338.005,E2 -15338.005} C_VEL
LIN {X 0,Y 319.563,Z 400.675,A -85,B 0,C 180,E1 -15341.606,E2 -15341.606} C_VEL
LIN {X 0,Y 319.486,Z 400.685,A -85,B 0,C 180,E1 -15345.258,E2 -15345.258} C_VEL
LIN {X 0,Y 319.526,Z 400.68,A -85,B 0,C 180,E1 -15348.713,E2 -15348.713} C_VEL
LIN {X 0,Y 319.553,Z 400.677,A -85,B 0,C 180,E1 -15352.35,E2 -15352.35} C_VEL
LIN {X 0,Y 319.559,Z 400.675,A -85,B 0,C 180,E1 -15355.124,E2 -15355.124} C_VEL
LIN {X 0,Y 319.566,Z 400.676,A -85,B 0,C 180,E1 -15359.06,E2 -15359.06} C_VEL
LIN {X 0,Y 319.606,Z 400.671,A -85,B 0,C 180,E1 -15362.499,E2 -15362.499} C_VEL
LIN {X 0,Y 319.605,Z 400.669,A -85,B 0,C 180,E1 -15365.305,E2 -15365.305} C_VEL
LIN {X 0,Y 319.598,Z 400.676,A -85,B 0,C 180,E1 -15368.049,E2 -15368.049} C_VEL
LIN {X 0,Y 319.691,Z 400.659,A -85,B 0,C 180,E1 -15370.963,E2 -15370.963} C_VEL
LIN {X 0,Y 319.733,Z 400.656,A -85,B 0,C 180,E1 -15375.276,E2 -15375.276} C_VEL
LIN {X 0,Y 319.761,Z 400.656,A -85,B 0,C 180,E1 -15379.873,E2 -15379.873} C_VEL
LIN {X 0,Y 319.937,Z 400.63,A -85,B 0,C 180,E1 -15382.427,E2 -15382.427} C_VEL
LIN {X 0,Y 319.955,Z 400.632,A -85,B 0,C 180,E1 -15383.695,E2 -15383.695} C_VEL
LIN {X 0,Y 319.964,Z 400.626,A -85,B 0,C 180,E1 -15388.742,E2 -15388.742} C_VEL
LIN {X 0,Y 318.988,Z 400.754,A -85,B 0,C 180,E1 -15391.263,E2 -15391.263} C_VEL
LIN {X 0,Y 319.079,Z 403.914,A -85,B 0,C 180,E1 -15395.055,E2 -15395.055} C_VEL
LIN {X 0,Y 318.928,Z 406.103,A -85,B 0,C 180,E1 -15397.598,E2 -15397.598} C_VEL
LIN {X 0,Y 318.766,Z 407.997,A -85,B 0,C 180,E1 -15399.718,E2 -15399.718} C_VEL
LIN {X 0,Y 323.09,Z 423.453,A -85,B 0,C 180,E1 -15400.766,E2 -15400.766} C_VEL
LIN {X 0,Y 325.915,Z 435.884,A -85,B 0,C 180,E1 -15401.821,E2 -15401.821} C_VEL
LIN {X 0,Y 326.671,Z 440.552,A -85,B 0,C 180,E1 -15402.266,E2 -15402.266} C_VEL
LIN {X 0,Y 325.599,Z 452.069,A -85,B 0,C 180,E1 -15403.378,E2 -15403.378} C_VEL
LIN {X 0,Y 324.314,Z 463.337,A -85,B 0,C 180,E1 -15404.751,E2 -15404.751} C_VEL
LIN {X 0,Y 323.146,Z 472.254,A -85,B 0,C 180,E1 -15406.099,E2 -15406.099} C_VEL
LIN {X 0,Y 321.914,Z 481.368,A -85,B 0,C 180,E1 -15407.797,E2 -15407.797} C_VEL
LIN {X 0,Y 320.782,Z 489.189,A -85,B 0,C 180,E1 -15409.594,E2 -15409.594} C_VEL
LIN {X 0,Y 319.862,Z 496.151,A -85,B 0,C 180,E1 -15411.594,E2 -15411.594} C_VEL
LIN {X 0,Y 319.237,Z 500.977,A -85,B 0,C 180,E1 -15413.345,E2 -15413.345} C_VEL
LIN {X 0,Y 318.678,Z 505.18,A -85,B 0,C 180,E1 -15415.283,E2 -15415.283} C_VEL
LIN {X 0,Y 318.226,Z 508.786,A -85,B 0,C 180,E1 -15417.631,E2 -15417.631} C_VEL
LIN {X 0,Y 317.996,Z 510.309,A -85,B 0,C 180,E1 -15419.092,E2 -15419.092} C_VEL
LIN {X 0,Y 317.894,Z 511.285,A -85,B 0,C 180,E1 -15420.563,E2 -15420.563} C_VEL
LIN {X 0,Y 317.89,Z 511.732,A -85,B 0,C 180,E1 -15422.847,E2 -15422.847} C_VEL
LIN {X 0,Y 318.097,Z 510.886,A -85,B 0,C 180,E1 -15425.167,E2 -15425.167} C_VEL
LIN {X 0,Y 318.488,Z 508.805,A -85,B 0,C 180,E1 -15427.4,E2 -15427.4} C_VEL
LIN {X 0,Y 319.107,Z 505.254,A -85,B 0,C 180,E1 -15429.694,E2 -15429.694} C_VEL
LIN {X 0,Y 319.773,Z 501.048,A -85,B 0,C 180,E1 -15431.646,E2 -15431.646} C_VEL
LIN {X 0,Y 320.712,Z 495.319,A -85,B 0,C 180,E1 -15433.684,E2 -15433.684} C_VEL
LIN {X 0,Y 321.939,Z 488.131,A -85,B 0,C 180,E1 -15435.687,E2 -15435.687} C_VEL
LIN {X 0,Y 323.396,Z 479.191,A -85,B 0,C 180,E1 -15437.636,E2 -15437.636} C_VEL
LIN {X 0,Y 324.773,Z 470.071,A -85,B 0,C 180,E1 -15439.234,E2 -15439.234} C_VEL
LIN {X 0,Y 326.182,Z 460.005,A -85,B 0,C 180,E1 -15440.653,E2 -15440.653} C_VEL
LIN {X 0,Y 327.451,Z 449.197,A -85,B 0,C 180,E1 -15441.871,E2 -15441.871} C_VEL
LIN {X 0,Y 328.114,Z 443.321,A -85,B 0,C 180,E1 -15442.42,E2 -15442.42} C_VEL
LIN {X 0,Y 326.886,Z 435.905,A -85,B 0,C 180,E1 -15443.179,E2 -15443.179} C_VEL
LIN {X 0,Y 323.373,Z 423.222,A -85,B 0,C 180,E1 -15444.352,E2 -15444.352} C_VEL
LIN {X 0,Y 319.419,Z 412.092,A -85,B 0,C 180,E1 -15445.249,E2 -15445.249} C_VEL
LIN {X 0,Y 318.884,Z 410.05,A -85,B 0,C 180,E1 -15445.399,E2 -15445.399} C_VEL
LIN {X 0,Y 319.124,Z 407.046,A -85,B 0,C 180,E1 -15449.232,E2 -15449.232} C_VEL
LIN {X 0,Y 319.309,Z 404.593,A -85,B 0,C 180,E1 -15452.47,E2 -15452.47} C_VEL
LIN {X 0,Y 319.441,Z 403.001,A -85,B 0,C 180,E1 -15454.655,E2 -15454.655} C_VEL
LIN {X 0,Y 318.787,Z 402.359,A -85,B 0,C 180,E1 -15455.701,E2 -15455.701} C_VEL
LIN {X 0,Y 315.941,Z 401.769,A -85,B 0,C 180,E1 -15457.413,E2 -15457.413} C_VEL
LIN {X 0,Y 313.563,Z 401.595,A -85,B 0,C 180,E1 -15458.804,E2 -15458.804} C_VEL
LIN {X 0,Y 312.604,Z 401.559,A -85,B 0,C 180,E1 -15459.881,E2 -15459.881} C_VEL
LIN {X 0,Y 312.559,Z 401.555,A -85,B 0,C 180,E1 -15460.245,E2 -15460.245} C_VEL
LIN {X 0,Y 312.603,Z 401.547,A -85,B 0,C 180,E1 -15463.006,E2 -15463.006} C_VEL
LIN {X 0,Y 312.69,Z 401.537,A -85,B 0,C 180,E1 -15465.686,E2 -15465.686} C_VEL
LIN {X 0,Y 312.694,Z 401.536,A -85,B 0,C 180,E1 -15469.641,E2 -15469.641} C_VEL
LIN {X 0,Y 312.849,Z 401.514,A -85,B 0,C 180,E1 -15472.254,E2 -15472.254} C_VEL
LIN {X 0,Y 312.711,Z 401.53,A -85,B 0,C 180,E1 -15474.842,E2 -15474.842} C_VEL
LIN {X 0,Y 312.986,Z 401.5,A -85,B 0,C 180,E1 -15478.713,E2 -15478.713} C_VEL
LIN {X 0,Y 312.988,Z 401.5,A -85,B 0,C 180,E1 -15481.287,E2 -15481.287} C_VEL
LIN {X 0,Y 312.711,Z 401.53,A -85,B 0,C 180,E1 -15485.158,E2 -15485.158} C_VEL
LIN {X 0,Y 312.849,Z 401.512,A -85,B 0,C 180,E1 -15487.746,E2 -15487.746} C_VEL
LIN {X 0,Y 312.665,Z 401.539,A -85,B 0,C 180,E1 -15491.671,E2 -15491.671} C_VEL
LIN {X 0,Y 312.696,Z 401.536,A -85,B 0,C 180,E1 -15494.888,E2 -15494.888} C_VEL
LIN {X 0,Y 312.628,Z 401.539,A -85,B 0,C 180,E1 -15499.237,E2 -15499.237} C_VEL
LIN {X 0,Y 312.542,Z 401.555,A -85,B 0,C 180,E1 -15502.789,E2 -15502.789} C_VEL
LIN {X 0,Y 312.593,Z 401.546,A -85,B 0,C 180,E1 -15505.933,E2 -15505.933} C_VEL
LIN {X 0,Y 312.535,Z 401.556,A -85,B 0,C 180,E1 -15509.651,E2 -15509.651} C_VEL
LIN {X 0,Y 312.517,Z 401.56,A -85,B 0,C 180,E1 -15513.689,E2 -15513.689} C_VEL
LIN {X 0,Y 312.549,Z 401.557,A -85,B 0,C 180,E1 -15517.382,E2 -15517.382} C_VEL
LIN {X 0,Y 312.613,Z 401.78,A -85,B 0,C 180,E1 -15518.493,E2 -15518.493} C_VEL
LIN {X 0,Y 313.252,Z 405.699,A -85,B 0,C 180,E1 -15522.304,E2 -15522.304} C_VEL
LIN {X 0,Y 314.038,Z 410.025,A -85,B 0,C 180,E1 -15526.072,E2 -15526.072} C_VEL
LIN {X 0,Y 314.886,Z 414.63,A -85,B 0,C 180,E1 -15529.665,E2 -15529.665} C_VEL
LIN {X 0,Y 315.384,Z 418.123,A -85,B 0,C 180,E1 -15532.208,E2 -15532.208} C_VEL
LIN {X 0,Y 315.468,Z 419.76,A -85,B 0,C 180,E1 -15533.322,E2 -15533.322} C_VEL
LIN {X 0,Y 314.807,Z 424.051,A -85,B 0,C 180,E1 -15536.074,E2 -15536.074} C_VEL
LIN {X 0,Y 313.828,Z 430.099,A -85,B 0,C 180,E1 -15539.744,E2 -15539.744} C_VEL
LIN {X 0,Y 312.828,Z 437.363,A -85,B 0,C 180,E1 -15543.98,E2 -15543.98} C_VEL
LIN {X 0,Y 312.402,Z 440.99,A -85,B 0,C 180,E1 -15546.025,E2 -15546.025} C_VEL
LIN {X 0,Y 315.706,Z 455.653,A -85,B 0,C 180,E1 -15546.979,E2 -15546.979} C_VEL
LIN {X 0,Y 317.473,Z 467.418,A -85,B 0,C 180,E1 -15547.893,E2 -15547.893} C_VEL
LIN {X 0,Y 318.397,Z 479.324,A -85,B 0,C 180,E1 -15548.992,E2 -15548.992} C_VEL
LIN {X 0,Y 318.736,Z 490.056,A -85,B 0,C 180,E1 -15550.183,E2 -15550.183} C_VEL
LIN {X 0,Y 317.008,Z 501.26,A -85,B 0,C 180,E1 -15551.584,E2 -15551.584} C_VEL
LIN {X 0,Y 315.467,Z 511.242,A -85,B 0,C 180,E1 -15553.165,E2 -15553.165} C_VEL
LIN {X 0,Y 314.29,Z 519.474,A -85,B 0,C 180,E1 -15554.767,E2 -15554.767} C_VEL
LIN {X 0,Y 313.039,Z 527.587,A -85,B 0,C 180,E1 -15556.696,E2 -15556.696} C_VEL
LIN {X 0,Y 312.16,Z 533.12,A -85,B 0,C 180,E1 -15558.309,E2 -15558.309} C_VEL
LIN {X 0,Y 311.519,Z 538.568,A -85,B 0,C 180,E1 -15560.258,E2 -15560.258} C_VEL
LIN {X 0,Y 311.064,Z 542.838,A -85,B 0,C 180,E1 -15562.209,E2 -15562.209} C_VEL
LIN {X 0,Y 310.909,Z 545.888,A -85,B 0,C 180,E1 -15564.047,E2 -15564.047} C_VEL
LIN {X 0,Y 310.844,Z 548.284,A -85,B 0,C 180,E1 -15566.11,E2 -15566.11} C_VEL
LIN {X 0,Y 310.852,Z 549.836,A -85,B 0,C 180,E1 -15568.704,E2 -15568.704} C_VEL
LIN {X 0,Y 310.975,Z 549.974,A -85,B 0,C 180,E1 -15570,E2 -15570} C_VEL
LIN {X 0,Y 310.885,Z 549.703,A -85,B 0,C 180,E1 -15571.295,E2 -15571.295} C_VEL
LIN {X 0,Y 310.847,Z 547.972,A -85,B 0,C 180,E1 -15573.889,E2 -15573.889} C_VEL
LIN {X 0,Y 310.908,Z 545.371,A -85,B 0,C 180,E1 -15575.95,E2 -15575.95} C_VEL
LIN {X 0,Y 311.064,Z 542.086,A -85,B 0,C 180,E1 -15577.791,E2 -15577.791} C_VEL
LIN {X 0,Y 311.521,Z 537.544,A -85,B 0,C 180,E1 -15579.741,E2 -15579.741} C_VEL
LIN {X 0,Y 312.291,Z 530.64,A -85,B 0,C 180,E1 -15582.014,E2 -15582.014} C_VEL
LIN {X 0,Y 313.407,Z 523.165,A -85,B 0,C 180,E1 -15583.949,E2 -15583.949} C_VEL
LIN {X 0,Y 314.65,Z 514.495,A -85,B 0,C 180,E1 -15585.757,E2 -15585.757} C_VEL
LIN {X 0,Y 315.872,Z 504.164,A -85,B 0,C 180,E1 -15587.479,E2 -15587.479} C_VEL
LIN {X 0,Y 317.353,Z 493.475,A -85,B 0,C 180,E1 -15588.897,E2 -15588.897} C_VEL
LIN {X 0,Y 318.095,Z 487.871,A -85,B 0,C 180,E1 -15589.521,E2 -15589.521} C_VEL
LIN {X 0,Y 317.216,Z 475.678,A -85,B 0,C 180,E1 -15590.761,E2 -15590.761} C_VEL
LIN {X 0,Y 315.752,Z 462.858,A -85,B 0,C 180,E1 -15591.808,E2 -15591.808} C_VEL
LIN {X 0,Y 313.649,Z 449.754,A -85,B 0,C 180,E1 -15592.641,E2 -15592.641} C_VEL
LIN {X 0,Y 312.289,Z 442.47,A -85,B 0,C 180,E1 -15593.024,E2 -15593.024} C_VEL
LIN {X 0,Y 312.995,Z 435.922,A -85,B 0,C 180,E1 -15596.684,E2 -15596.684} C_VEL
LIN {X 0,Y 313.78,Z 429.663,A -85,B 0,C 180,E1 -15600.261,E2 -15600.261} C_VEL
LIN {X 0,Y 314.856,Z 422.75,A -85,B 0,C 180,E1 -15604.321,E2 -15604.321} C_VEL
LIN {X 0,Y 315.355,Z 418.391,A -85,B 0,C 180,E1 -15606.992,E2 -15606.992} C_VEL
LIN {X 0,Y 314.886,Z 414.548,A -85,B 0,C 180,E1 -15609.499,E2 -15609.499} C_VEL
LIN {X 0,Y 313.881,Z 409.12,A -85,B 0,C 180,E1 -15613.267,E2 -15613.267} C_VEL
LIN {X 0,Y 313.059,Z 404.382,A -85,B 0,C 180,E1 -15616.787,E2 -15616.787} C_VEL
LIN {X 0,Y 312.519,Z 401.558,A -85,B 0,C 180,E1 -15619.083,E2 -15619.083} C_VEL
LIN {X 0,Y 312.536,Z 401.555,A -85,B 0,C 180,E1 -15622.616,E2 -15622.616} C_VEL
LIN {X 0,Y 312.514,Z 401.555,A -85,B 0,C 180,E1 -15626.31,E2 -15626.31} C_VEL
LIN {X 0,Y 312.532,Z 401.553,A -85,B 0,C 180,E1 -15630.349,E2 -15630.349} C_VEL
LIN {X 0,Y 312.59,Z 401.545,A -85,B 0,C 180,E1 -15634.066,E2 -15634.066} C_VEL
LIN {X 0,Y 312.581,Z 401.546,A -85,B 0,C 180,E1 -15637.528,E2 -15637.528} C_VEL
LIN {X 0,Y 312.631,Z 401.539,A -85,B 0,C 180,E1 -15641.656,E2 -15641.656} C_VEL
LIN {X 0,Y 312.686,Z 401.532,A -85,B 0,C 180,E1 -15645.686,E2 -15645.686} C_VEL
LIN {X 0,Y 312.691,Z 401.532,A -85,B 0,C 180,E1 -15649.642,E2 -15649.642} C_VEL
LIN {X 0,Y 312.846,Z 401.514,A -85,B 0,C 180,E1 -15652.254,E2 -15652.254} C_VEL
LIN {X 0,Y 312.709,Z 401.533,A -85,B 0,C 180,E1 -15654.842,E2 -15654.842} C_VEL
LIN {X 0,Y 312.985,Z 401.5,A -85,B 0,C 180,E1 -15658.713,E2 -15658.713} C_VEL
LIN {X 0,Y 313.113,Z 401.48,A -85,B 0,C 180,E1 -15660,E2 -15660} C_VEL
LIN {X 0,Y 312.93,Z 401.506,A -85,B 0,C 180,E1 -15662.575,E2 -15662.575} C_VEL
LIN {X 0,Y 312.887,Z 401.51,A -85,B 0,C 180,E1 -15666.632,E2 -15666.632} C_VEL
LIN {X 0,Y 312.781,Z 401.522,A -85,B 0,C 180,E1 -15669.05,E2 -15669.05} C_VEL
LIN {X 0,Y 312.627,Z 401.539,A -85,B 0,C 180,E1 -15672.992,E2 -15672.992} C_VEL
LIN {X 0,Y 312.631,Z 401.539,A -85,B 0,C 180,E1 -15675.65,E2 -15675.65} C_VEL
LIN {X 0,Y 312.624,Z 401.54,A -85,B 0,C 180,E1 -15679.237,E2 -15679.237} C_VEL
LIN {X 0,Y 312.539,Z 401.551,A -85,B 0,C 180,E1 -15682.79,E2 -15682.79} C_VEL
LIN {X 0,Y 312.597,Z 401.545,A -85,B 0,C 180,E1 -15685.936,E2 -15685.936} C_VEL
LIN {X 0,Y 312.54,Z 401.551,A -85,B 0,C 180,E1 -15689.651,E2 -15689.651} C_VEL
LIN {X 0,Y 312.515,Z 401.553,A -85,B 0,C 180,E1 -15693.69,E2 -15693.69} C_VEL
LIN {X 0,Y 312.537,Z 401.551,A -85,B 0,C 180,E1 -15697.384,E2 -15697.384} C_VEL
LIN {X 0,Y 312.496,Z 401.556,A -85,B 0,C 180,E1 -15700.709,E2 -15700.709} C_VEL
LIN {X 0,Y 312.452,Z 401.567,A -85,B 0,C 180,E1 -15704.21,E2 -15704.21} C_VEL
LIN {X 0,Y 312.482,Z 401.561,A -85,B 0,C 180,E1 -15707.92,E2 -15707.92} C_VEL
LIN {X 0,Y 312.497,Z 401.552,A -85,B 0,C 180,E1 -15710.972,E2 -15710.972} C_VEL
LIN {X 0,Y 312.531,Z 401.554,A -85,B 0,C 180,E1 -15714.221,E2 -15714.221} C_VEL
LIN {X 0,Y 312.504,Z 401.556,A -85,B 0,C 180,E1 -15717.335,E2 -15717.335} C_VEL
LIN {X 0,Y 312.544,Z 401.551,A -85,B 0,C 180,E1 -15721.28,E2 -15721.28} C_VEL
LIN {X 0,Y 312.586,Z 401.543,A -85,B 0,C 180,E1 -15724.712,E2 -15724.712} C_VEL
LIN {X 0,Y 312.589,Z 401.546,A -85,B 0,C 180,E1 -15727.53,E2 -15727.53} C_VEL
LIN {X 0,Y 312.64,Z 401.541,A -85,B 0,C 180,E1 -15731.657,E2 -15731.657} C_VEL
LIN {X 0,Y 312.696,Z 401.535,A -85,B 0,C 180,E1 -15735.687,E2 -15735.687} C_VEL
LIN {X 0,Y 312.705,Z 401.533,A -85,B 0,C 180,E1 -15739.642,E2 -15739.642} C_VEL
LIN {X 0,Y 312.875,Z 401.511,A -85,B 0,C 180,E1 -15742.255,E2 -15742.255} C_VEL
LIN {X 0,Y 312.913,Z 401.508,A -85,B 0,C 180,E1 -15743.553,E2 -15743.553} C_VEL
LIN {X 0,Y 312.931,Z 401.502,A -85,B 0,C 180,E1 -15748.713,E2 -15748.713} C_VEL
LIN {X 0,Y 311.941,Z 401.691,A -85,B 0,C 180,E1 -15751.291,E2 -15751.291} C_VEL
LIN {X 0,Y 312.039,Z 403.826,A -85,B 0,C 180,E1 -15753.875,E2 -15753.875} C_VEL
LIN {X 0,Y 311.905,Z 406.916,A -85,B 0,C 180,E1 -15757.504,E2 -15757.504} C_VEL
LIN {X 0,Y 311.762,Z 408.67,A -85,B 0,C 180,E1 -15759.284,E2 -15759.284} C_VEL
LIN {X 0,Y 315.509,Z 421.677,A -85,B 0,C 180,E1 -15760.154,E2 -15760.154} C_VEL
LIN {X 0,Y 318.392,Z 433.557,A -85,B 0,C 180,E1 -15761.148,E2 -15761.148} C_VEL
LIN {X 0,Y 319.868,Z 441.847,A -85,B 0,C 180,E1 -15761.957,E2 -15761.957} C_VEL
LIN {X 0,Y 318.732,Z 453.4,A -85,B 0,C 180,E1 -15763.114,E2 -15763.114} C_VEL
LIN {X 0,Y 317.48,Z 463.81,A -85,B 0,C 180,E1 -15764.421,E2 -15764.421} C_VEL
LIN {X 0,Y 316.274,Z 472.717,A -85,B 0,C 180,E1 -15765.796,E2 -15765.796} C_VEL
LIN {X 0,Y 314.988,Z 481.827,A -85,B 0,C 180,E1 -15767.53,E2 -15767.53} C_VEL
LIN {X 0,Y 313.881,Z 489.325,A -85,B 0,C 180,E1 -15769.285,E2 -15769.285} C_VEL
LIN {X 0,Y 312.843,Z 496.607,A -85,B 0,C 180,E1 -15771.411,E2 -15771.411} C_VEL
LIN {X 0,Y 312.198,Z 501.544,A -85,B 0,C 180,E1 -15773.247,E2 -15773.247} C_VEL
LIN {X 0,Y 311.558,Z 506.239,A -85,B 0,C 180,E1 -15775.536,E2 -15775.536} C_VEL
LIN {X 0,Y 311.336,Z 508.26,A -85,B 0,C 180,E1 -15776.838,E2 -15776.838} C_VEL
LIN {X 0,Y 311.034,Z 510.073,A -85,B 0,C 180,E1 -15778.327,E2 -15778.327} C_VEL
LIN {X 0,Y 310.818,Z 511.8,A -85,B 0,C 180,E1 -15780.769,E2 -15780.769} C_VEL
LIN {X 0,Y 310.832,Z 512.144,A -85,B 0,C 180,E1 -15783.219,E2 -15783.219} C_VEL
LIN {X 0,Y 311.084,Z 511.137,A -85,B 0,C 180,E1 -15785.579,E2 -15785.579} C_VEL
LIN {X 0,Y 311.53,Z 508.868,A -85,B 0,C 180,E1 -15787.853,E2 -15787.853} C_VEL
LIN {X 0,Y 312.128,Z 505.452,A -85,B 0,C 180,E1 -15790.043,E2 -15790.043} C_VEL
LIN {X 0,Y 312.983,Z 500.423,A -85,B 0,C 180,E1 -15792.348,E2 -15792.348} C_VEL
LIN {X 0,Y 314.131,Z 494.125,A -85,B 0,C 180,E1 -15794.502,E2 -15794.502} C_VEL
LIN {X 0,Y 315.559,Z 486.052,A -85,B 0,C 180,E1 -15796.645,E2 -15796.645} C_VEL
LIN {X 0,Y 316.899,Z 478.28,A -85,B 0,C 180,E1 -15798.292,E2 -15798.292} C_VEL
LIN {X 0,Y 318.371,Z 468.645,A -85,B 0,C 180,E1 -15799.947,E2 -15799.947} C_VEL
LIN {X 0,Y 319.939,Z 457.297,A -85,B 0,C 180,E1 -15801.495,E2 -15801.495} C_VEL
LIN {X 0,Y 321.267,Z 446.516,A -85,B 0,C 180,E1 -15802.654,E2 -15802.654} C_VEL
LIN {X 0,Y 321.342,Z 442.72,A -85,B 0,C 180,E1 -15803.026,E2 -15803.026} C_VEL
LIN {X 0,Y 318.928,Z 432.083,A -85,B 0,C 180,E1 -15804.148,E2 -15804.148} C_VEL
LIN {X 0,Y 315.226,Z 420.052,A -85,B 0,C 180,E1 -15805.255,E2 -15805.255} C_VEL
LIN {X 0,Y 311.905,Z 410.521,A -85,B 0,C 180,E1 -15806.042,E2 -15806.042} C_VEL
LIN {X 0,Y 312.071,Z 408.374,A -85,B 0,C 180,E1 -15808.845,E2 -15808.845} C_VEL
LIN {X 0,Y 312.264,Z 406.179,A -85,B 0,C 180,E1 -15811.794,E2 -15811.794} C_VEL
LIN {X 0,Y 312.428,Z 404.078,A -85,B 0,C 180,E1 -15814.697,E2 -15814.697} C_VEL
LIN {X 0,Y 312.524,Z 402.125,A -85,B 0,C 180,E1 -15817.524,E2 -15817.524} C_VEL
LIN {X 0,Y 312.499,Z 401.565,A -85,B 0,C 180,E1 -15818.91,E2 -15818.91} C_VEL
LIN {X 0,Y 312.559,Z 401.555,A -85,B 0,C 180,E1 -15820.245,E2 -15820.245} C_VEL
LIN {X 0,Y 311.989,Z 401.63,A -85,B 0,C 180,E1 -15821.321,E2 -15821.321} C_VEL
LIN {X 0,Y 309.202,Z 401.977,A -85,B 0,C 180,E1 -15823.075,E2 -15823.075} C_VEL
LIN {X 0,Y 306.768,Z 402.275,A -85,B 0,C 180,E1 -15824.496,E2 -15824.496} C_VEL
LIN {X 0,Y 305.695,Z 402.408,A -85,B 0,C 180,E1 -15825.597,E2 -15825.597} C_VEL
LIN {X 0,Y 305.596,Z 402.417,A -85,B 0,C 180,E1 -15825.97,E2 -15825.97} C_VEL
LIN {X 0,Y 305.632,Z 402.416,A -85,B 0,C 180,E1 -15829.399,E2 -15829.399} C_VEL
LIN {X 0,Y 305.793,Z 402.394,A -85,B 0,C 180,E1 -15832.074,E2 -15832.074} C_VEL
LIN {X 0,Y 305.683,Z 402.405,A -85,B 0,C 180,E1 -15834.723,E2 -15834.723} C_VEL
LIN {X 0,Y 305.953,Z 402.376,A -85,B 0,C 180,E1 -15838.684,E2 -15838.684} C_VEL
LIN {X 0,Y 305.955,Z 402.376,A -85,B 0,C 180,E1 -15841.316,E2 -15841.316} C_VEL
LIN {X 0,Y 305.838,Z 402.39,A -85,B 0,C 180,E1 -15846.598,E2 -15846.598} C_VEL
LIN {X 0,Y 305.7,Z 402.407,A -85,B 0,C 180,E1 -15849.261,E2 -15849.261} C_VEL
LIN {X 0,Y 305.584,Z 402.416,A -85,B 0,C 180,E1 -15853.296,E2 -15853.296} C_VEL
LIN {X 0,Y 305.59,Z 402.415,A -85,B 0,C 180,E1 -15856.02,E2 -15856.02} C_VEL
LIN {X 0,Y 305.574,Z 402.419,A -85,B 0,C 180,E1 -15859.445,E2 -15859.445} C_VEL
LIN {X 0,Y 305.487,Z 402.434,A -85,B 0,C 180,E1 -15863.041,E2 -15863.041} C_VEL
LIN {X 0,Y 305.522,Z 402.425,A -85,B 0,C 180,E1 -15866.219,E2 -15866.219} C_VEL
LIN {X 0,Y 305.484,Z 402.431,A -85,B 0,C 180,E1 -15869.047,E2 -15869.047} C_VEL
LIN {X 0,Y 305.439,Z 402.443,A -85,B 0,C 180,E1 -15871.953,E2 -15871.953} C_VEL
LIN {X 0,Y 305.46,Z 402.439,A -85,B 0,C 180,E1 -15875.114,E2 -15875.114} C_VEL
LIN {X 0,Y 305.545,Z 402.549,A -85,B 0,C 180,E1 -15877.556,E2 -15877.556} C_VEL
LIN {X 0,Y 306.201,Z 406.617,A -85,B 0,C 180,E1 -15881.73,E2 -15881.73} C_VEL
LIN {X 0,Y 306.878,Z 410.474,A -85,B 0,C 180,E1 -15885.231,E2 -15885.231} C_VEL
LIN {X 0,Y 307.714,Z 414.957,A -85,B 0,C 180,E1 -15888.912,E2 -15888.912} C_VEL
LIN {X 0,Y 308.373,Z 419.122,A -85,B 0,C 180,E1 -15892.023,E2 -15892.023} C_VEL
LIN {X 0,Y 308.368,Z 421.458,A -85,B 0,C 180,E1 -15893.661,E2 -15893.661} C_VEL
LIN {X 0,Y 307.542,Z 426.219,A -85,B 0,C 180,E1 -15896.739,E2 -15896.739} C_VEL
LIN {X 0,Y 306.538,Z 432.469,A -85,B 0,C 180,E1 -15900.602,E2 -15900.602} C_VEL
LIN {X 0,Y 305.716,Z 438.34,A -85,B 0,C 180,E1 -15904.101,E2 -15904.101} C_VEL
LIN {X 0,Y 305.479,Z 440.538,A -85,B 0,C 180,E1 -15905.378,E2 -15905.378} C_VEL
LIN {X 0,Y 308.708,Z 454.442,A -85,B 0,C 180,E1 -15906.304,E2 -15906.304} C_VEL
LIN {X 0,Y 310.656,Z 466.657,A -85,B 0,C 180,E1 -15907.293,E2 -15907.293} C_VEL
LIN {X 0,Y 311.676,Z 479.695,A -85,B 0,C 180,E1 -15908.544,E2 -15908.544} C_VEL
LIN {X 0,Y 312.011,Z 490.053,A -85,B 0,C 180,E1 -15909.738,E2 -15909.738} C_VEL
LIN {X 0,Y 310.27,Z 501.146,A -85,B 0,C 180,E1 -15911.169,E2 -15911.169} C_VEL
LIN {X 0,Y 308.656,Z 511.072,A -85,B 0,C 180,E1 -15912.782,E2 -15912.782} C_VEL
LIN {X 0,Y 307.433,Z 519.259,A -85,B 0,C 180,E1 -15914.419,E2 -15914.419} C_VEL
LIN {X 0,Y 306.089,Z 527.331,A -85,B 0,C 180,E1 -15916.388,E2 -15916.388} C_VEL
LIN {X 0,Y 305.171,Z 532.822,A -85,B 0,C 180,E1 -15918.038,E2 -15918.038} C_VEL
LIN {X 0,Y 304.478,Z 538.234,A -85,B 0,C 180,E1 -15920.031,E2 -15920.031} C_VEL
LIN {X 0,Y 304.016,Z 542.477,A -85,B 0,C 180,E1 -15922.027,E2 -15922.027} C_VEL
LIN {X 0,Y 303.831,Z 545.733,A -85,B 0,C 180,E1 -15924.07,E2 -15924.07} C_VEL
LIN {X 0,Y 303.753,Z 547.884,A -85,B 0,C 180,E1 -15926.02,E2 -15926.02} C_VEL
LIN {X 0,Y 303.708,Z 548.852,A -85,B 0,C 180,E1 -15927.347,E2 -15927.347} C_VEL
LIN {X 0,Y 303.76,Z 549.41,A -85,B 0,C 180,E1 -15928.674,E2 -15928.674} C_VEL
LIN {X 0,Y 303.886,Z 549.536,A -85,B 0,C 180,E1 -15930,E2 -15930} C_VEL
LIN {X 0,Y 303.792,Z 549.256,A -85,B 0,C 180,E1 -15931.325,E2 -15931.325} C_VEL
LIN {X 0,Y 303.717,Z 548.581,A -85,B 0,C 180,E1 -15932.652,E2 -15932.652} C_VEL
LIN {X 0,Y 303.779,Z 547.499,A -85,B 0,C 180,E1 -15933.979,E2 -15933.979} C_VEL
LIN {X 0,Y 303.839,Z 545.091,A -85,B 0,C 180,E1 -15935.945,E2 -15935.945} C_VEL
LIN {X 0,Y 304.016,Z 541.574,A -85,B 0,C 180,E1 -15937.972,E2 -15937.972} C_VEL
LIN {X 0,Y 304.48,Z 537.003,A -85,B 0,C 180,E1 -15939.968,E2 -15939.968} C_VEL
LIN {X 0,Y 305.285,Z 530.06,A -85,B 0,C 180,E1 -15942.294,E2 -15942.294} C_VEL
LIN {X 0,Y 306.448,Z 522.553,A -85,B 0,C 180,E1 -15944.272,E2 -15944.272} C_VEL
LIN {X 0,Y 307.783,Z 513.556,A -85,B 0,C 180,E1 -15946.17,E2 -15946.17} C_VEL
LIN {X 0,Y 309.037,Z 503.448,A -85,B 0,C 180,E1 -15947.879,E2 -15947.879} C_VEL
LIN {X 0,Y 310.645,Z 492.71,A -85,B 0,C 180,E1 -15949.321,E2 -15949.321} C_VEL
LIN {X 0,Y 311.145,Z 487.011,A -85,B 0,C 180,E1 -15949.976,E2 -15949.976} C_VEL
LIN {X 0,Y 310.202,Z 474.651,A -85,B 0,C 180,E1 -15951.253,E2 -15951.253} C_VEL
LIN {X 0,Y 308.703,Z 461.655,A -85,B 0,C 180,E1 -15952.327,E2 -15952.327} C_VEL
LIN {X 0,Y 306.496,Z 448.668,A -85,B 0,C 180,E1 -15953.161,E2 -15953.161} C_VEL
LIN {X 0,Y 305.275,Z 442.064,A -85,B 0,C 180,E1 -15953.515,E2 -15953.515} C_VEL
LIN {X 0,Y 306.024,Z 435.439,A -85,B 0,C 180,E1 -15957.342,E2 -15957.342} C_VEL
LIN {X 0,Y 306.847,Z 429.173,A -85,B 0,C 180,E1 -15961.019,E2 -15961.019} C_VEL
LIN {X 0,Y 307.906,Z 422.961,A -85,B 0,C 180,E1 -15964.793,E2 -15964.793} C_VEL
LIN {X 0,Y 308.319,Z 419.299,A -85,B 0,C 180,E1 -15967.078,E2 -15967.078} C_VEL
LIN {X 0,Y 307.801,Z 415.363,A -85,B 0,C 180,E1 -15969.74,E2 -15969.74} C_VEL
LIN {X 0,Y 306.888,Z 410.215,A -85,B 0,C 180,E1 -15973.394,E2 -15973.394} C_VEL
LIN {X 0,Y 305.959,Z 405.061,A -85,B 0,C 180,E1 -15977.31,E2 -15977.31} C_VEL
LIN {X 0,Y 305.474,Z 402.434,A -85,B 0,C 180,E1 -15979.505,E2 -15979.505} C_VEL
LIN {X 0,Y 305.492,Z 402.433,A -85,B 0,C 180,E1 -15983.263,E2 -15983.263} C_VEL
LIN {X 0,Y 305.459,Z 402.435,A -85,B 0,C 180,E1 -15986.483,E2 -15986.483} C_VEL
LIN {X 0,Y 305.452,Z 402.435,A -85,B 0,C 180,E1 -15989.59,E2 -15989.59} C_VEL
LIN {X 0,Y 305.508,Z 402.43,A -85,B 0,C 180,E1 -15992.607,E2 -15992.607} C_VEL
LIN {X 0,Y 305.501,Z 402.428,A -85,B 0,C 180,E1 -15995.538,E2 -15995.538} C_VEL
LIN {X 0,Y 305.513,Z 402.426,A -85,B 0,C 180,E1 -15999.815,E2 -15999.815} C_VEL
LIN {X 0,Y 305.567,Z 402.423,A -85,B 0,C 180,E1 -16002.603,E2 -16002.603} C_VEL
LIN {X 0,Y 305.642,Z 402.411,A -85,B 0,C 180,E1 -16005.349,E2 -16005.349} C_VEL
LIN {X 0,Y 305.628,Z 402.412,A -85,B 0,C 180,E1 -16009.399,E2 -16009.399} C_VEL
LIN {X 0,Y 305.789,Z 402.392,A -85,B 0,C 180,E1 -16012.074,E2 -16012.074} C_VEL
LIN {X 0,Y 305.68,Z 402.408,A -85,B 0,C 180,E1 -16014.723,E2 -16014.723} C_VEL
LIN {X 0,Y 305.952,Z 402.376,A -85,B 0,C 180,E1 -16018.684,E2 -16018.684} C_VEL
LIN {X 0,Y 305.952,Z 402.371,A -85,B 0,C 180,E1 -16021.316,E2 -16021.316} C_VEL
LIN {X 0,Y 305.843,Z 402.39,A -85,B 0,C 180,E1 -16026.61,E2 -16026.61} C_VEL
LIN {X 0,Y 305.729,Z 402.399,A -85,B 0,C 180,E1 -16029.26,E2 -16029.26} C_VEL
LIN {X 0,Y 305.581,Z 402.415,A -85,B 0,C 180,E1 -16033.297,E2 -16033.297} C_VEL
LIN {X 0,Y 305.587,Z 402.418,A -85,B 0,C 180,E1 -16036.021,E2 -16036.021} C_VEL
LIN {X 0,Y 305.571,Z 402.419,A -85,B 0,C 180,E1 -16039.446,E2 -16039.446} C_VEL
LIN {X 0,Y 305.484,Z 402.428,A -85,B 0,C 180,E1 -16043.042,E2 -16043.042} C_VEL
LIN {X 0,Y 305.542,Z 402.426,A -85,B 0,C 180,E1 -16046.228,E2 -16046.228} C_VEL
LIN {X 0,Y 305.49,Z 402.429,A -85,B 0,C 180,E1 -16049.051,E2 -16049.051} C_VEL
LIN {X 0,Y 305.46,Z 402.431,A -85,B 0,C 180,E1 -16053.518,E2 -16053.518} C_VEL
LIN {X 0,Y 305.493,Z 402.43,A -85,B 0,C 180,E1 -16056.737,E2 -16056.737} C_VEL
LIN {X 0,Y 305.461,Z 402.436,A -85,B 0,C 180,E1 -16060.108,E2 -16060.108} C_VEL
LIN {X 0,Y 305.431,Z 402.437,A -85,B 0,C 180,E1 -16063.654,E2 -16063.654} C_VEL
LIN {X 0,Y 305.452,Z 402.434,A -85,B 0,C 180,E1 -16067.415,E2 -16067.415} C_VEL
LIN {X 0,Y 305.466,Z 402.428,A -85,B 0,C 180,E1 -16071.597,E2 -16071.597} C_VEL
LIN {X 0,Y 305.461,Z 402.431,A -85,B 0,C 180,E1 -16074.888,E2 -16074.888} C_VEL
LIN {X 0,Y 305.45,Z 402.437,A -85,B 0,C 180,E1 -16078.356,E2 -16078.356} C_VEL
LIN {X 0,Y 305.513,Z 402.426,A -85,B 0,C 180,E1 -16081.114,E2 -16081.114} C_VEL
LIN {X 0,Y 305.572,Z 402.419,A -85,B 0,C 180,E1 -16084.089,E2 -16084.089} C_VEL
LIN {X 0,Y 305.502,Z 402.429,A -85,B 0,C 180,E1 -16088.404,E2 -16088.404} C_VEL
LIN {X 0,Y 305.592,Z 402.416,A -85,B 0,C 180,E1 -16091.219,E2 -16091.219} C_VEL
LIN {X 0,Y 305.651,Z 402.41,A -85,B 0,C 180,E1 -16095.35,E2 -16095.35} C_VEL
LIN {X 0,Y 305.641,Z 402.411,A -85,B 0,C 180,E1 -16099.4,E2 -16099.4} C_VEL
LIN {X 0,Y 305.816,Z 402.392,A -85,B 0,C 180,E1 -16102.075,E2 -16102.075} C_VEL
LIN {X 0,Y 305.669,Z 402.406,A -85,B 0,C 180,E1 -16104.724,E2 -16104.724} C_VEL
LIN {X 0,Y 305.898,Z 402.378,A -85,B 0,C 180,E1 -16108.684,E2 -16108.684} C_VEL
LIN {X 0,Y 304.896,Z 402.635,A -85,B 0,C 180,E1 -16111.321,E2 -16111.321} C_VEL
LIN {X 0,Y 305.001,Z 404.771,A -85,B 0,C 180,E1 -16113.964,E2 -16113.964} C_VEL
LIN {X 0,Y 304.806,Z 408.188,A -85,B 0,C 180,E1 -16117.952,E2 -16117.952} C_VEL
LIN {X 0,Y 304.728,Z 408.891,A -85,B 0,C 180,E1 -16118.774,E2 -16118.774} C_VEL
LIN {X 0,Y 308.72,Z 422.95,A -85,B 0,C 180,E1 -16119.755,E2 -16119.755} C_VEL
LIN {X 0,Y 311.517,Z 434.514,A -85,B 0,C 180,E1 -16120.76,E2 -16120.76} C_VEL
LIN {X 0,Y 313.008,Z 441.9,A -85,B 0,C 180,E1 -16121.511,E2 -16121.511} C_VEL
LIN {X 0,Y 312.003,Z 453.388,A -85,B 0,C 180,E1 -16122.687,E2 -16122.687} C_VEL
LIN {X 0,Y 310.75,Z 463.551,A -85,B 0,C 180,E1 -16123.976,E2 -16123.976} C_VEL
LIN {X 0,Y 309.429,Z 473.157,A -85,B 0,C 180,E1 -16125.478,E2 -16125.478} C_VEL
LIN {X 0,Y 308.087,Z 482.271,A -85,B 0,C 180,E1 -16127.251,E2 -16127.251} C_VEL
LIN {X 0,Y 306.769,Z 490.719,A -85,B 0,C 180,E1 -16129.294,E2 -16129.294} C_VEL
LIN {X 0,Y 305.84,Z 497.054,A -85,B 0,C 180,E1 -16131.218,E2 -16131.218} C_VEL
LIN {X 0,Y 305.184,Z 501.87,A -85,B 0,C 180,E1 -16133.047,E2 -16133.047} C_VEL
LIN {X 0,Y 304.538,Z 506.238,A -85,B 0,C 180,E1 -16135.168,E2 -16135.168} C_VEL
LIN {X 0,Y 304.083,Z 509.669,A -85,B 0,C 180,E1 -16137.532,E2 -16137.532} C_VEL
LIN {X 0,Y 303.838,Z 511.192,A -85,B 0,C 180,E1 -16139.061,E2 -16139.061} C_VEL
LIN {X 0,Y 303.705,Z 512.365,A -85,B 0,C 180,E1 -16141.105,E2 -16141.105} C_VEL
LIN {X 0,Y 303.77,Z 512.499,A -85,B 0,C 180,E1 -16143.728,E2 -16143.728} C_VEL
LIN {X 0,Y 304.063,Z 511.344,A -85,B 0,C 180,E1 -16146.003,E2 -16146.003} C_VEL
LIN {X 0,Y 304.653,Z 508.676,A -85,B 0,C 180,E1 -16148.525,E2 -16148.525} C_VEL
LIN {X 0,Y 305.419,Z 504.262,A -85,B 0,C 180,E1 -16151.128,E2 -16151.128} C_VEL
LIN {X 0,Y 306.463,Z 498.666,A -85,B 0,C 180,E1 -16153.47,E2 -16153.47} C_VEL
LIN {X 0,Y 307.705,Z 492.209,A -85,B 0,C 180,E1 -16155.54,E2 -16155.54} C_VEL
LIN {X 0,Y 309.219,Z 483.879,A -85,B 0,C 180,E1 -16157.626,E2 -16157.626} C_VEL
LIN {X 0,Y 310.849,Z 474.656,A -85,B 0,C 180,E1 -16159.468,E2 -16159.468} C_VEL
LIN {X 0,Y 312.372,Z 464.904,A -85,B 0,C 180,E1 -16161.024,E2 -16161.024} C_VEL
LIN {X 0,Y 313.811,Z 454.554,A -85,B 0,C 180,E1 -16162.352,E2 -16162.352} C_VEL
LIN {X 0,Y 314.912,Z 445.407,A -85,B 0,C 180,E1 -16163.306,E2 -16163.306} C_VEL
LIN {X 0,Y 312.762,Z 435.177,A -85,B 0,C 180,E1 -16164.448,E2 -16164.448} C_VEL
LIN {X 0,Y 309.272,Z 423.368,A -85,B 0,C 180,E1 -16165.62,E2 -16165.62} C_VEL
LIN {X 0,Y 305.455,Z 413.046,A -85,B 0,C 180,E1 -16166.531,E2 -16166.531} C_VEL
LIN {X 0,Y 304.937,Z 411.007,A -85,B 0,C 180,E1 -16166.714,E2 -16166.714} C_VEL
LIN {X 0,Y 305.189,Z 407.777,A -85,B 0,C 180,E1 -16171.079,E2 -16171.079} C_VEL
LIN {X 0,Y 305.37,Z 405.648,A -85,B 0,C 180,E1 -16174.069,E2 -16174.069} C_VEL
LIN {X 0,Y 305.489,Z 403.671,A -85,B 0,C 180,E1 -16176.977,E2 -16176.977} C_VEL
LIN {X 0,Y 305.472,Z 402.74,A -85,B 0,C 180,E1 -16178.401,E2 -16178.401} C_VEL
LIN {X 0,Y 305.575,Z 402.424,A -85,B 0,C 180,E1 -16181.216,E2 -16181.216} C_VEL
LIN {X 0,Y 305.645,Z 402.414,A -85,B 0,C 180,E1 -16185.349,E2 -16185.349} C_VEL
LIN {X 0,Y 305.596,Z 402.417,A -85,B 0,C 180,E1 -16185.97,E2 -16185.97} C_VEL
LIN {X 0,Y 304.909,Z 402.506,A -85,B 0,C 180,E1 -16187.069,E2 -16187.069} C_VEL
LIN {X 0,Y 302.104,Z 402.853,A -85,B 0,C 180,E1 -16188.862,E2 -16188.862} C_VEL
LIN {X 0,Y 299.767,Z 403.144,A -85,B 0,C 180,E1 -16190.315,E2 -16190.315} C_VEL
LIN {X 0,Y 298.797,Z 403.267,A -85,B 0,C 180,E1 -16191.439,E2 -16191.439} C_VEL
LIN {X 0,Y 298.734,Z 403.274,A -85,B 0,C 180,E1 -16191.819,E2 -16191.819} C_VEL
LIN {X 0,Y 298.653,Z 403.281,A -85,B 0,C 180,E1 -16194.599,E2 -16194.599} C_VEL
LIN {X 0,Y 298.919,Z 403.252,A -85,B 0,C 180,E1 -16198.653,E2 -16198.653} C_VEL
LIN {X 0,Y 298.921,Z 403.252,A -85,B 0,C 180,E1 -16201.347,E2 -16201.347} C_VEL
LIN {X 0,Y 298.783,Z 403.268,A -85,B 0,C 180,E1 -16206.754,E2 -16206.754} C_VEL
LIN {X 0,Y 298.632,Z 403.287,A -85,B 0,C 180,E1 -16209.482,E2 -16209.482} C_VEL
LIN {X 0,Y 298.548,Z 403.292,A -85,B 0,C 180,E1 -16213.615,E2 -16213.615} C_VEL
LIN {X 0,Y 298.545,Z 403.293,A -85,B 0,C 180,E1 -16216.409,E2 -16216.409} C_VEL
LIN {X 0,Y 298.509,Z 403.3,A -85,B 0,C 180,E1 -16219.655,E2 -16219.655} C_VEL
LIN {X 0,Y 298.454,Z 403.309,A -85,B 0,C 180,E1 -16223.598,E2 -16223.598} C_VEL
LIN {X 0,Y 298.482,Z 403.302,A -85,B 0,C 180,E1 -16226.575,E2 -16226.575} C_VEL
LIN {X 0,Y 298.413,Z 403.315,A -85,B 0,C 180,E1 -16229.642,E2 -16229.642} C_VEL
LIN {X 0,Y 298.392,Z 403.318,A -85,B 0,C 180,E1 -16232.801,E2 -16232.801} C_VEL
LIN {X 0,Y 298.482,Z 403.437,A -85,B 0,C 180,E1 -16236.695,E2 -16236.695} C_VEL
LIN {X 0,Y 298.895,Z 405.872,A -85,B 0,C 180,E1 -16239.41,E2 -16239.41} C_VEL
LIN {X 0,Y 299.552,Z 409.853,A -85,B 0,C 180,E1 -16243.339,E2 -16243.339} C_VEL
LIN {X 0,Y 300.384,Z 414.331,A -85,B 0,C 180,E1 -16247.274,E2 -16247.274} C_VEL
LIN {X 0,Y 301.167,Z 418.917,A -85,B 0,C 180,E1 -16250.945,E2 -16250.945} C_VEL
LIN {X 0,Y 301.438,Z 421.255,A -85,B 0,C 180,E1 -16252.686,E2 -16252.686} C_VEL
LIN {X 0,Y 301.107,Z 424.294,A -85,B 0,C 180,E1 -16254.778,E2 -16254.778} C_VEL
LIN {X 0,Y 299.906,Z 430.756,A -85,B 0,C 180,E1 -16258.966,E2 -16258.966} C_VEL
LIN {X 0,Y 298.992,Z 436.831,A -85,B 0,C 180,E1 -16262.72,E2 -16262.72} C_VEL
LIN {X 0,Y 298.557,Z 440.219,A -85,B 0,C 180,E1 -16264.686,E2 -16264.686} C_VEL
LIN {X 0,Y 301.949,Z 454.548,A -85,B 0,C 180,E1 -16265.697,E2 -16265.697} C_VEL
LIN {X 0,Y 303.928,Z 466.342,A -85,B 0,C 180,E1 -16266.699,E2 -16266.699} C_VEL
LIN {X 0,Y 304.911,Z 479.157,A -85,B 0,C 180,E1 -16267.965,E2 -16267.965} C_VEL
LIN {X 0,Y 305.241,Z 490.094,A -85,B 0,C 180,E1 -16269.268,E2 -16269.268} C_VEL
LIN {X 0,Y 303.767,Z 499.963,A -85,B 0,C 180,E1 -16270.574,E2 -16270.574} C_VEL
LIN {X 0,Y 302.172,Z 509.112,A -85,B 0,C 180,E1 -16272.051,E2 -16272.051} C_VEL
LIN {X 0,Y 300.872,Z 517.546,A -85,B 0,C 180,E1 -16273.722,E2 -16273.722} C_VEL
LIN {X 0,Y 299.406,Z 525.831,A -85,B 0,C 180,E1 -16275.731,E2 -16275.731} C_VEL
LIN {X 0,Y 298.19,Z 532.537,A -85,B 0,C 180,E1 -16277.753,E2 -16277.753} C_VEL
LIN {X 0,Y 297.454,Z 537.92,A -85,B 0,C 180,E1 -16279.793,E2 -16279.793} C_VEL
LIN {X 0,Y 296.963,Z 542.135,A -85,B 0,C 180,E1 -16281.836,E2 -16281.836} C_VEL
LIN {X 0,Y 296.739,Z 545.621,A -85,B 0,C 180,E1 -16284.119,E2 -16284.119} C_VEL
LIN {X 0,Y 296.665,Z 547.488,A -85,B 0,C 180,E1 -16285.924,E2 -16285.924} C_VEL
LIN {X 0,Y 296.631,Z 548.446,A -85,B 0,C 180,E1 -16287.284,E2 -16287.284} C_VEL
LIN {X 0,Y 296.668,Z 548.982,A -85,B 0,C 180,E1 -16288.642,E2 -16288.642} C_VEL
LIN {X 0,Y 296.797,Z 549.099,A -85,B 0,C 180,E1 -16290,E2 -16290} C_VEL
LIN {X 0,Y 296.7,Z 548.808,A -85,B 0,C 180,E1 -16291.357,E2 -16291.357} C_VEL
LIN {X 0,Y 296.641,Z 548.124,A -85,B 0,C 180,E1 -16292.716,E2 -16292.716} C_VEL
LIN {X 0,Y 296.69,Z 547.02,A -85,B 0,C 180,E1 -16294.075,E2 -16294.075} C_VEL
LIN {X 0,Y 296.738,Z 544.875,A -85,B 0,C 180,E1 -16295.88,E2 -16295.88} C_VEL
LIN {X 0,Y 296.963,Z 541.054,A -85,B 0,C 180,E1 -16298.163,E2 -16298.163} C_VEL
LIN {X 0,Y 297.456,Z 536.452,A -85,B 0,C 180,E1 -16300.206,E2 -16300.206} C_VEL
LIN {X 0,Y 298.312,Z 529.466,A -85,B 0,C 180,E1 -16302.586,E2 -16302.586} C_VEL
LIN {X 0,Y 299.494,Z 521.917,A -85,B 0,C 180,E1 -16304.611,E2 -16304.611} C_VEL
LIN {X 0,Y 300.728,Z 514.217,A -85,B 0,C 180,E1 -16306.286,E2 -16306.286} C_VEL
LIN {X 0,Y 301.948,Z 504.827,A -85,B 0,C 180,E1 -16307.962,E2 -16307.962} C_VEL
LIN {X 0,Y 303.498,Z 494.443,A -85,B 0,C 180,E1 -16309.443,E2 -16309.443} C_VEL
LIN {X 0,Y 304.285,Z 489.033,A -85,B 0,C 180,E1 -16310.093,E2 -16310.093} C_VEL
LIN {X 0,Y 303.456,Z 476.572,A -85,B 0,C 180,E1 -16311.479,E2 -16311.479} C_VEL
LIN {X 0,Y 302.084,Z 463.768,A -85,B 0,C 180,E1 -16312.607,E2 -16312.607} C_VEL
LIN {X 0,Y 299.988,Z 450.674,A -85,B 0,C 180,E1 -16313.524,E2 -16313.524} C_VEL
LIN {X 0,Y 298.274,Z 441.705,A -85,B 0,C 180,E1 -16314.027,E2 -16314.027} C_VEL
LIN {X 0,Y 299.091,Z 434.944,A -85,B 0,C 180,E1 -16318.031,E2 -16318.031} C_VEL
LIN {X 0,Y 299.798,Z 429.967,A -85,B 0,C 180,E1 -16321.045,E2 -16321.045} C_VEL
LIN {X 0,Y 300.965,Z 423.303,A -85,B 0,C 180,E1 -16325.184,E2 -16325.184} C_VEL
LIN {X 0,Y 301.256,Z 419.716,A -85,B 0,C 180,E1 -16327.516,E2 -16327.516} C_VEL
LIN {X 0,Y 300.51,Z 414.855,A -85,B 0,C 180,E1 -16330.906,E2 -16330.906} C_VEL
LIN {X 0,Y 299.603,Z 409.719,A -85,B 0,C 180,E1 -16334.725,E2 -16334.725} C_VEL
LIN {X 0,Y 298.645,Z 404.541,A -85,B 0,C 180,E1 -16338.854,E2 -16338.854} C_VEL
LIN {X 0,Y 298.424,Z 403.313,A -85,B 0,C 180,E1 -16339.884,E2 -16339.884} C_VEL
LIN {X 0,Y 298.427,Z 403.31,A -85,B 0,C 180,E1 -16343.931,E2 -16343.931} C_VEL
LIN {X 0,Y 298.388,Z 403.315,A -85,B 0,C 180,E1 -16347.983,E2 -16347.983} C_VEL
LIN {X 0,Y 298.451,Z 403.307,A -85,B 0,C 180,E1 -16351.903,E2 -16351.903} C_VEL
LIN {X 0,Y 298.477,Z 403.307,A -85,B 0,C 180,E1 -16354.923,E2 -16354.923} C_VEL
LIN {X 0,Y 298.444,Z 403.308,A -85,B 0,C 180,E1 -16359.315,E2 -16359.315} C_VEL
LIN {X 0,Y 298.531,Z 403.297,A -85,B 0,C 180,E1 -16362.179,E2 -16362.179} C_VEL
LIN {X 0,Y 298.586,Z 403.292,A -85,B 0,C 180,E1 -16364.994,E2 -16364.994} C_VEL
LIN {X 0,Y 298.584,Z 403.291,A -85,B 0,C 180,E1 -16369.146,E2 -16369.146} C_VEL
LIN {X 0,Y 298.733,Z 403.27,A -85,B 0,C 180,E1 -16371.885,E2 -16371.885} C_VEL
LIN {X 0,Y 298.65,Z 403.283,A -85,B 0,C 180,E1 -16374.599,E2 -16374.599} C_VEL
LIN {X 0,Y 298.918,Z 403.253,A -85,B 0,C 180,E1 -16378.653,E2 -16378.653} C_VEL
LIN {X 0,Y 298.918,Z 403.247,A -85,B 0,C 180,E1 -16381.347,E2 -16381.347} C_VEL
LIN {X 0,Y 298.79,Z 403.267,A -85,B 0,C 180,E1 -16386.754,E2 -16386.754} C_VEL
LIN {X 0,Y 298.674,Z 403.278,A -85,B 0,C 180,E1 -16389.481,E2 -16389.481} C_VEL
LIN {X 0,Y 298.545,Z 403.291,A -85,B 0,C 180,E1 -16393.616,E2 -16393.616} C_VEL
LIN {X 0,Y 298.542,Z 403.299,A -85,B 0,C 180,E1 -16396.409,E2 -16396.409} C_VEL
LIN {X 0,Y 298.506,Z 403.299,A -85,B 0,C 180,E1 -16399.655,E2 -16399.655} C_VEL
LIN {X 0,Y 298.451,Z 403.303,A -85,B 0,C 180,E1 -16403.598,E2 -16403.598} C_VEL
LIN {X 0,Y 298.484,Z 403.305,A -85,B 0,C 180,E1 -16406.575,E2 -16406.575} C_VEL
LIN {X 0,Y 298.416,Z 403.31,A -85,B 0,C 180,E1 -16409.642,E2 -16409.642} C_VEL
LIN {X 0,Y 298.391,Z 403.312,A -85,B 0,C 180,E1 -16412.801,E2 -16412.801} C_VEL
LIN {X 0,Y 298.462,Z 403.306,A -85,B 0,C 180,E1 -16416.814,E2 -16416.814} C_VEL
LIN {X 0,Y 298.414,Z 403.308,A -85,B 0,C 180,E1 -16421.095,E2 -16421.095} C_VEL
LIN {X 0,Y 298.423,Z 403.309,A -85,B 0,C 180,E1 -16423.11,E2 -16423.11} C_VEL
LIN {X 0,Y 298.4,Z 403.312,A -85,B 0,C 180,E1 -16426.922,E2 -16426.922} C_VEL
LIN {X 0,Y 298.397,Z 403.307,A -85,B 0,C 180,E1 -16431.008,E2 -16431.008} C_VEL
LIN {X 0,Y 298.417,Z 403.307,A -85,B 0,C 180,E1 -16433.931,E2 -16433.931} C_VEL
LIN {X 0,Y 298.394,Z 403.318,A -85,B 0,C 180,E1 -16437.985,E2 -16437.985} C_VEL
LIN {X 0,Y 298.459,Z 403.309,A -85,B 0,C 180,E1 -16441.905,E2 -16441.905} C_VEL
LIN {X 0,Y 298.486,Z 403.297,A -85,B 0,C 180,E1 -16444.925,E2 -16444.925} C_VEL
LIN {X 0,Y 298.452,Z 403.307,A -85,B 0,C 180,E1 -16449.316,E2 -16449.316} C_VEL
LIN {X 0,Y 298.54,Z 403.294,A -85,B 0,C 180,E1 -16452.18,E2 -16452.18} C_VEL
LIN {X 0,Y 298.596,Z 403.288,A -85,B 0,C 180,E1 -16454.996,E2 -16454.996} C_VEL
LIN {X 0,Y 298.596,Z 403.287,A -85,B 0,C 180,E1 -16459.147,E2 -16459.147} C_VEL
LIN {X 0,Y 298.762,Z 403.272,A -85,B 0,C 180,E1 -16461.887,E2 -16461.887} C_VEL
LIN {X 0,Y 298.643,Z 403.282,A -85,B 0,C 180,E1 -16464.599,E2 -16464.599} C_VEL
LIN {X 0,Y 298.863,Z 403.255,A -85,B 0,C 180,E1 -16468.653,E2 -16468.653} C_VEL
LIN {X 0,Y 297.853,Z 403.605,A -85,B 0,C 180,E1 -16471.352,E2 -16471.352} C_VEL
LIN {X 0,Y 297.963,Z 405.732,A -85,B 0,C 180,E1 -16474.058,E2 -16474.058} C_VEL
LIN {X 0,Y 297.802,Z 408.685,A -85,B 0,C 180,E1 -16477.612,E2 -16477.612} C_VEL
LIN {X 0,Y 297.754,Z 409.392,A -85,B 0,C 180,E1 -16478.268,E2 -16478.268} C_VEL
LIN {X 0,Y 301.494,Z 422.535,A -85,B 0,C 180,E1 -16479.202,E2 -16479.202} C_VEL
LIN {X 0,Y 304.414,Z 434.148,A -85,B 0,C 180,E1 -16480.236,E2 -16480.236} C_VEL
LIN {X 0,Y 306.267,Z 443.835,A -85,B 0,C 180,E1 -16481.248,E2 -16481.248} C_VEL
LIN {X 0,Y 305.07,Z 455.317,A -85,B 0,C 180,E1 -16482.473,E2 -16482.473} C_VEL
LIN {X 0,Y 303.744,Z 465.481,A -85,B 0,C 180,E1 -16483.835,E2 -16483.835} C_VEL
LIN {X 0,Y 302.286,Z 475.512,A -85,B 0,C 180,E1 -16485.508,E2 -16485.508} C_VEL
LIN {X 0,Y 300.942,Z 483.944,A -85,B 0,C 180,E1 -16487.237,E2 -16487.237} C_VEL
LIN {X 0,Y 299.749,Z 491.56,A -85,B 0,C 180,E1 -16489.162,E2 -16489.162} C_VEL
LIN {X 0,Y 298.685,Z 498.502,A -85,B 0,C 180,E1 -16491.39,E2 -16491.39} C_VEL
LIN {X 0,Y 297.862,Z 503.953,A -85,B 0,C 180,E1 -16493.648,E2 -16493.648} C_VEL
LIN {X 0,Y 297.336,Z 508.29,A -85,B 0,C 180,E1 -16496.078,E2 -16496.078} C_VEL
LIN {X 0,Y 296.795,Z 511.431,A -85,B 0,C 180,E1 -16498.818,E2 -16498.818} C_VEL
LIN {X 0,Y 296.614,Z 512.919,A -85,B 0,C 180,E1 -16501.461,E2 -16501.461} C_VEL
LIN {X 0,Y 296.723,Z 512.88,A -85,B 0,C 180,E1 -16504.004,E2 -16504.004} C_VEL
LIN {X 0,Y 297.057,Z 511.552,A -85,B 0,C 180,E1 -16506.447,E2 -16506.447} C_VEL
LIN {X 0,Y 297.646,Z 509.015,A -85,B 0,C 180,E1 -16508.813,E2 -16508.813} C_VEL
LIN {X 0,Y 298.392,Z 504.982,A -85,B 0,C 180,E1 -16511.26,E2 -16511.26} C_VEL
LIN {X 0,Y 299.312,Z 500.421,A -85,B 0,C 180,E1 -16513.289,E2 -16513.289} C_VEL
LIN {X 0,Y 300.546,Z 494.171,A -85,B 0,C 180,E1 -16515.45,E2 -16515.45} C_VEL
LIN {X 0,Y 302.1,Z 486.365,A -85,B 0,C 180,E1 -16517.573,E2 -16517.573} C_VEL
LIN {X 0,Y 303.807,Z 477.233,A -85,B 0,C 180,E1 -16519.521,E2 -16519.521} C_VEL
LIN {X 0,Y 305.45,Z 467.388,A -85,B 0,C 180,E1 -16521.207,E2 -16521.207} C_VEL
LIN {X 0,Y 307.117,Z 456.283,A -85,B 0,C 180,E1 -16522.714,E2 -16522.714} C_VEL
LIN {X 0,Y 308.238,Z 447.839,A -85,B 0,C 180,E1 -16523.643,E2 -16523.643} C_VEL
LIN {X 0,Y 307.685,Z 443.284,A -85,B 0,C 180,E1 -16524.174,E2 -16524.174} C_VEL
LIN {X 0,Y 305.143,Z 432.777,A -85,B 0,C 180,E1 -16525.367,E2 -16525.367} C_VEL
LIN {X 0,Y 301.463,Z 421.205,A -85,B 0,C 180,E1 -16526.53,E2 -16526.53} C_VEL
LIN {X 0,Y 298.038,Z 412.055,A -85,B 0,C 180,E1 -16527.344,E2 -16527.344} C_VEL
LIN {X 0,Y 297.937,Z 411.514,A -85,B 0,C 180,E1 -16527.408,E2 -16527.408} C_VEL
LIN {X 0,Y 298.198,Z 408.298,A -85,B 0,C 180,E1 -16531.877,E2 -16531.877} C_VEL
LIN {X 0,Y 298.384,Z 406.215,A -85,B 0,C 180,E1 -16534.915,E2 -16534.915} C_VEL
LIN {X 0,Y 298.478,Z 404.275,A -85,B 0,C 180,E1 -16537.868,E2 -16537.868} C_VEL
LIN {X 0,Y 298.424,Z 403.386,A -85,B 0,C 180,E1 -16539.313,E2 -16539.313} C_VEL
LIN {X 0,Y 298.531,Z 403.301,A -85,B 0,C 180,E1 -16542.179,E2 -16542.179} C_VEL
LIN {X 0,Y 298.542,Z 403.297,A -85,B 0,C 180,E1 -16545.969,E2 -16545.969} C_VEL
LIN {X 0,Y 298.632,Z 403.285,A -85,B 0,C 180,E1 -16550.518,E2 -16550.518} C_VEL
LIN {X 0,Y 298.734,Z 403.274,A -85,B 0,C 180,E1 -16551.819,E2 -16551.819} C_VEL
LIN {X 0,Y 298.106,Z 403.354,A -85,B 0,C 180,E1 -16552.943,E2 -16552.943} C_VEL
LIN {X 0,Y 295.267,Z 403.705,A -85,B 0,C 180,E1 -16554.773,E2 -16554.773} C_VEL
LIN {X 0,Y 292.862,Z 404.007,A -85,B 0,C 180,E1 -16556.258,E2 -16556.258} C_VEL
LIN {X 0,Y 291.866,Z 404.126,A -85,B 0,C 180,E1 -16557.408,E2 -16557.408} C_VEL
LIN {X 0,Y 291.806,Z 404.133,A -85,B 0,C 180,E1 -16557.797,E2 -16557.797} C_VEL
LIN {X 0,Y 291.961,Z 404.114,A -85,B 0,C 180,E1 -16560,E2 -16560} C_VEL
LIN {X 0,Y 291.785,Z 404.136,A -85,B 0,C 180,E1 -16562.761,E2 -16562.761} C_VEL
LIN {X 0,Y 291.732,Z 404.147,A -85,B 0,C 180,E1 -16566.918,E2 -16566.918} C_VEL
LIN {X 0,Y 291.571,Z 404.166,A -85,B 0,C 180,E1 -16569.714,E2 -16569.714} C_VEL
LIN {X 0,Y 291.518,Z 404.169,A -85,B 0,C 180,E1 -16573.95,E2 -16573.95} C_VEL
LIN {X 0,Y 291.484,Z 404.174,A -85,B 0,C 180,E1 -16576.818,E2 -16576.818} C_VEL
LIN {X 0,Y 291.448,Z 404.181,A -85,B 0,C 180,E1 -16579.875,E2 -16579.875} C_VEL
LIN {X 0,Y 291.396,Z 404.189,A -85,B 0,C 180,E1 -16584.206,E2 -16584.206} C_VEL
LIN {X 0,Y 291.416,Z 404.185,A -85,B 0,C 180,E1 -16587.272,E2 -16587.272} C_VEL
LIN {X 0,Y 291.331,Z 404.197,A -85,B 0,C 180,E1 -16590.438,E2 -16590.438} C_VEL
LIN {X 0,Y 291.342,Z 404.198,A -85,B 0,C 180,E1 -16593.699,E2 -16593.699} C_VEL
LIN {X 0,Y 291.391,Z 404.338,A -85,B 0,C 180,E1 -16595.795,E2 -16595.795} C_VEL
LIN {X 0,Y 292.011,Z 407.678,A -85,B 0,C 180,E1 -16599.632,E2 -16599.632} C_VEL
LIN {X 0,Y 292.758,Z 412.188,A -85,B 0,C 180,E1 -16604.121,E2 -16604.121} C_VEL
LIN {X 0,Y 293.559,Z 416.458,A -85,B 0,C 180,E1 -16607.916,E2 -16607.916} C_VEL
LIN {X 0,Y 294.314,Z 421.051,A -85,B 0,C 180,E1 -16611.622,E2 -16611.622} C_VEL
LIN {X 0,Y 294.22,Z 424.759,A -85,B 0,C 180,E1 -16614.307,E2 -16614.307} C_VEL
LIN {X 0,Y 293.082,Z 430.508,A -85,B 0,C 180,E1 -16618.16,E2 -16618.16} C_VEL
LIN {X 0,Y 292.095,Z 436.509,A -85,B 0,C 180,E1 -16622.019,E2 -16622.019} C_VEL
LIN {X 0,Y 291.641,Z 439.554,A -85,B 0,C 180,E1 -16623.916,E2 -16623.916} C_VEL
LIN {X 0,Y 295.141,Z 454.066,A -85,B 0,C 180,E1 -16625.007,E2 -16625.007} C_VEL
LIN {X 0,Y 297.275,Z 466.783,A -85,B 0,C 180,E1 -16626.145,E2 -16626.145} C_VEL
